LIN {X 0,Y 573.232,Z 251.703,A -85,B 0,C 180,E1 -2309.118,E2 -2309.118} C_VEL
LIN {X 0,Y 573.231,Z 251.702,A -85,B 0,C 180,E1 -2311.435,E2 -2311.435} C_VEL
LIN {X 0,Y 573.254,Z 251.705,A -85,B 0,C 180,E1 -2314.59,E2 -2314.59} C_VEL
LIN {X 0,Y 573.236,Z 251.705,A -85,B 0,C 180,E1 -2317.662,E2 -2317.662} C_VEL
LIN {X 0,Y 573.276,Z 251.851,A -85,B 0,C 180,E1 -2318.673,E2 -2318.673} C_VEL
LIN {X 0,Y 573.837,Z 256.408,A -85,B 0,C 180,E1 -2319.383,E2 -2319.383} C_VEL
LIN {X 0,Y 573.742,Z 263.76,A -85,B 0,C 180,E1 -2320.45,E2 -2320.45} C_VEL
LIN {X 0,Y 575.209,Z 270.767,A -85,B 0,C 180,E1 -2320.593,E2 -2320.593} C_VEL
LIN {X 0,Y 574.754,Z 427.05,A -85,B 0,C 180,E1 -2322.612,E2 -2322.612} C_VEL
LIN {X 0,Y 574.651,Z 442.817,A -85,B 0,C 180,E1 -2322.954,E2 -2322.954} C_VEL
LIN {X 0,Y 574.452,Z 456.451,A -85,B 0,C 180,E1 -2323.382,E2 -2323.382} C_VEL
LIN {X 0,Y 574.308,Z 469.862,A -85,B 0,C 180,E1 -2323.926,E2 -2323.926} C_VEL
LIN {X 0,Y 574.101,Z 483.847,A -85,B 0,C 180,E1 -2324.649,E2 -2324.649} C_VEL
LIN {X 0,Y 573.911,Z 496.092,A -85,B 0,C 180,E1 -2325.413,E2 -2325.413} C_VEL
LIN {X 0,Y 573.693,Z 508.609,A -85,B 0,C 180,E1 -2326.36,E2 -2326.36} C_VEL
LIN {X 0,Y 573.571,Z 518.669,A -85,B 0,C 180,E1 -2327.258,E2 -2327.258} C_VEL
LIN {X 0,Y 573.399,Z 528.984,A -85,B 0,C 180,E1 -2328.332,E2 -2328.332} C_VEL
LIN {X 0,Y 573.267,Z 538.996,A -85,B 0,C 180,E1 -2329.582,E2 -2329.582} C_VEL
LIN {X 0,Y 573.137,Z 547.362,A -85,B 0,C 180,E1 -2330.827,E2 -2330.827} C_VEL
LIN {X 0,Y 573.081,Z 555.183,A -85,B 0,C 180,E1 -2332.247,E2 -2332.247} C_VEL
LIN {X 0,Y 573.03,Z 561.427,A -85,B 0,C 180,E1 -2333.662,E2 -2333.662} C_VEL
LIN {X 0,Y 572.95,Z 566.262,A -85,B 0,C 180,E1 -2335.074,E2 -2335.074} C_VEL
LIN {X 0,Y 573.006,Z 569.794,A -85,B 0,C 180,E1 -2336.484,E2 -2336.484} C_VEL
LIN {X 0,Y 572.933,Z 572.153,A -85,B 0,C 180,E1 -2337.891,E2 -2337.891} C_VEL
LIN {X 0,Y 572.937,Z 573.314,A -85,B 0,C 180,E1 -2339.297,E2 -2339.297} C_VEL
LIN {X 0,Y 572.939,Z 573.342,A -85,B 0,C 180,E1 -2340.702,E2 -2340.702} C_VEL
LIN {X 0,Y 572.937,Z 572.256,A -85,B 0,C 180,E1 -2342.108,E2 -2342.108} C_VEL
LIN {X 0,Y 573.007,Z 569.983,A -85,B 0,C 180,E1 -2343.515,E2 -2343.515} C_VEL
LIN {X 0,Y 572.952,Z 566.528,A -85,B 0,C 180,E1 -2344.925,E2 -2344.925} C_VEL
LIN {X 0,Y 573.017,Z 561.792,A -85,B 0,C 180,E1 -2346.337,E2 -2346.337} C_VEL
LIN {X 0,Y 573.072,Z 555.625,A -85,B 0,C 180,E1 -2347.752,E2 -2347.752} C_VEL
LIN {X 0,Y 573.135,Z 547.941,A -85,B 0,C 180,E1 -2349.172,E2 -2349.172} C_VEL
LIN {X 0,Y 573.265,Z 539.657,A -85,B 0,C 180,E1 -2350.417,E2 -2350.417} C_VEL
LIN {X 0,Y 573.354,Z 529.786,A -85,B 0,C 180,E1 -2351.668,E2 -2351.668} C_VEL
LIN {X 0,Y 573.533,Z 519.618,A -85,B 0,C 180,E1 -2352.742,E2 -2352.742} C_VEL
LIN {X 0,Y 573.694,Z 508.608,A -85,B 0,C 180,E1 -2353.73,E2 -2353.73} C_VEL
LIN {X 0,Y 573.916,Z 496.248,A -85,B 0,C 180,E1 -2354.667,E2 -2354.667} C_VEL
LIN {X 0,Y 574.088,Z 483.851,A -85,B 0,C 180,E1 -2355.441,E2 -2355.441} C_VEL
LIN {X 0,Y 574.302,Z 469.864,A -85,B 0,C 180,E1 -2356.164,E2 -2356.164} C_VEL
LIN {X 0,Y 574.468,Z 456.434,A -85,B 0,C 180,E1 -2356.707,E2 -2356.707} C_VEL
LIN {X 0,Y 574.632,Z 441.329,A -85,B 0,C 180,E1 -2357.178,E2 -2357.178} C_VEL
LIN {X 0,Y 574.721,Z 432.945,A -85,B 0,C 180,E1 -2357.369,E2 -2357.369} C_VEL
LIN {X 0,Y 574.195,Z 427.214,A -85,B 0,C 180,E1 -2357.501,E2 -2357.501} C_VEL
LIN {X 0,Y 568.693,Z 408.639,A -85,B 0,C 180,E1 -2357.931,E2 -2357.931} C_VEL
LIN {X 0,Y 568.057,Z 402.835,A -85,B 0,C 180,E1 -2358.024,E2 -2358.024} C_VEL
LIN {X 0,Y 568.401,Z 270.982,A -85,B 0,C 180,E1 -2359.737,E2 -2359.737} C_VEL
LIN {X 0,Y 566.817,Z 263.453,A -85,B 0,C 180,E1 -2359.902,E2 -2359.902} C_VEL
LIN {X 0,Y 566.779,Z 255.764,A -85,B 0,C 180,E1 -2361.075,E2 -2361.075} C_VEL
LIN {X 0,Y 566.19,Z 252.586,A -85,B 0,C 180,E1 -2361.605,E2 -2361.605} C_VEL
LIN {X 0,Y 566.175,Z 252.587,A -85,B 0,C 180,E1 -2364.181,E2 -2364.181} C_VEL
LIN {X 0,Y 566.185,Z 252.579,A -85,B 0,C 180,E1 -2366.653,E2 -2366.653} C_VEL
LIN {X 0,Y 566.177,Z 252.579,A -85,B 0,C 180,E1 -2368.953,E2 -2368.953} C_VEL
LIN {X 0,Y 566.189,Z 252.58,A -85,B 0,C 180,E1 -2371.421,E2 -2371.421} C_VEL
LIN {X 0,Y 566.208,Z 252.584,A -85,B 0,C 180,E1 -2373.955,E2 -2373.955} C_VEL
LIN {X 0,Y 566.181,Z 252.579,A -85,B 0,C 180,E1 -2376.57,E2 -2376.57} C_VEL
LIN {X 0,Y 566.213,Z 252.581,A -85,B 0,C 180,E1 -2379.685,E2 -2379.685} C_VEL
LIN {X 0,Y 566.198,Z 252.576,A -85,B 0,C 180,E1 -2382.916,E2 -2382.916} C_VEL
LIN {X 0,Y 566.191,Z 252.583,A -85,B 0,C 180,E1 -2386.048,E2 -2386.048} C_VEL
LIN {X 0,Y 566.201,Z 252.577,A -85,B 0,C 180,E1 -2389.213,E2 -2389.213} C_VEL
LIN {X 0,Y 566.182,Z 252.586,A -85,B 0,C 180,E1 -2391.636,E2 -2391.636} C_VEL
LIN {X 0,Y 566.16,Z 252.583,A -85,B 0,C 180,E1 -2394.307,E2 -2394.307} C_VEL
LIN {X 0,Y 566.2,Z 252.576,A -85,B 0,C 180,E1 -2396.896,E2 -2396.896} C_VEL
LIN {X 0,Y 566.175,Z 252.584,A -85,B 0,C 180,E1 -2399.406,E2 -2399.406} C_VEL
LIN {X 0,Y 566.181,Z 252.586,A -85,B 0,C 180,E1 -2401.855,E2 -2401.855} C_VEL
LIN {X 0,Y 566.2,Z 252.578,A -85,B 0,C 180,E1 -2404.25,E2 -2404.25} C_VEL
LIN {X 0,Y 566.163,Z 252.58,A -85,B 0,C 180,E1 -2406.718,E2 -2406.718} C_VEL
LIN {X 0,Y 566.202,Z 252.586,A -85,B 0,C 180,E1 -2409.662,E2 -2409.662} C_VEL
LIN {X 0,Y 566.192,Z 252.577,A -85,B 0,C 180,E1 -2412.667,E2 -2412.667} C_VEL
LIN {X 0,Y 566.221,Z 252.583,A -85,B 0,C 180,E1 -2415.626,E2 -2415.626} C_VEL
LIN {X 0,Y 566.228,Z 252.572,A -85,B 0,C 180,E1 -2418.674,E2 -2418.674} C_VEL
LIN {X 0,Y 566.223,Z 252.58,A -85,B 0,C 180,E1 -2421.433,E2 -2421.433} C_VEL
LIN {X 0,Y 566.244,Z 252.571,A -85,B 0,C 180,E1 -2424.301,E2 -2424.301} C_VEL
LIN {X 0,Y 566.268,Z 252.571,A -85,B 0,C 180,E1 -2427.153,E2 -2427.153} C_VEL
LIN {X 0,Y 566.273,Z 252.57,A -85,B 0,C 180,E1 -2429.999,E2 -2429.999} C_VEL
LIN {X 0,Y 566.262,Z 252.569,A -85,B 0,C 180,E1 -2432.845,E2 -2432.845} C_VEL
LIN {X 0,Y 566.249,Z 252.577,A -85,B 0,C 180,E1 -2435.697,E2 -2435.697} C_VEL
LIN {X 0,Y 566.195,Z 252.576,A -85,B 0,C 180,E1 -2438.565,E2 -2438.565} C_VEL
LIN {X 0,Y 566.231,Z 252.582,A -85,B 0,C 180,E1 -2441.453,E2 -2441.453} C_VEL
LIN {X 0,Y 566.218,Z 252.573,A -85,B 0,C 180,E1 -2444.504,E2 -2444.504} C_VEL
LIN {X 0,Y 566.187,Z 252.585,A -85,B 0,C 180,E1 -2447.331,E2 -2447.331} C_VEL
LIN {X 0,Y 566.2,Z 252.576,A -85,B 0,C 180,E1 -2450.336,E2 -2450.336} C_VEL
LIN {X 0,Y 566.159,Z 252.589,A -85,B 0,C 180,E1 -2453.281,E2 -2453.281} C_VEL
LIN {X 0,Y 566.2,Z 252.58,A -85,B 0,C 180,E1 -2455.748,E2 -2455.748} C_VEL
LIN {X 0,Y 566.189,Z 252.577,A -85,B 0,C 180,E1 -2458.201,E2 -2458.201} C_VEL
LIN {X 0,Y 566.186,Z 252.583,A -85,B 0,C 180,E1 -2461.077,E2 -2461.077} C_VEL
LIN {X 0,Y 566.198,Z 252.58,A -85,B 0,C 180,E1 -2463.734,E2 -2463.734} C_VEL
LIN {X 0,Y 566.194,Z 252.577,A -85,B 0,C 180,E1 -2466.569,E2 -2466.569} C_VEL
LIN {X 0,Y 566.198,Z 252.58,A -85,B 0,C 180,E1 -2469.685,E2 -2469.685} C_VEL
LIN {X 0,Y 566.175,Z 252.579,A -85,B 0,C 180,E1 -2472.089,E2 -2472.089} C_VEL
LIN {X 0,Y 566.159,Z 252.587,A -85,B 0,C 180,E1 -2475.035,E2 -2475.035} C_VEL
LIN {X 0,Y 566.175,Z 252.58,A -85,B 0,C 180,E1 -2477.91,E2 -2477.91} C_VEL
LIN {X 0,Y 566.206,Z 252.577,A -85,B 0,C 180,E1 -2480.727,E2 -2480.727} C_VEL
LIN {X 0,Y 566.188,Z 252.579,A -85,B 0,C 180,E1 -2483.785,E2 -2483.785} C_VEL
LIN {X 0,Y 566.197,Z 252.576,A -85,B 0,C 180,E1 -2486.266,E2 -2486.266} C_VEL
LIN {X 0,Y 566.184,Z 252.583,A -85,B 0,C 180,E1 -2488.922,E2 -2488.922} C_VEL
LIN {X 0,Y 566.196,Z 252.577,A -85,B 0,C 180,E1 -2491.857,E2 -2491.857} C_VEL
LIN {X 0,Y 566.199,Z 252.576,A -85,B 0,C 180,E1 -2494.251,E2 -2494.251} C_VEL
LIN {X 0,Y 566.158,Z 252.584,A -85,B 0,C 180,E1 -2496.718,E2 -2496.718} C_VEL
LIN {X 0,Y 566.203,Z 252.578,A -85,B 0,C 180,E1 -2499.663,E2 -2499.663} C_VEL
LIN {X 0,Y 566.184,Z 252.581,A -85,B 0,C 180,E1 -2502.669,E2 -2502.669} C_VEL
LIN {X 0,Y 566.214,Z 252.576,A -85,B 0,C 180,E1 -2505.627,E2 -2505.627} C_VEL
LIN {X 0,Y 566.22,Z 252.577,A -85,B 0,C 180,E1 -2508.676,E2 -2508.676} C_VEL
LIN {X 0,Y 566.193,Z 252.581,A -85,B 0,C 180,E1 -2511.434,E2 -2511.434} C_VEL
LIN {X 0,Y 566.246,Z 252.571,A -85,B 0,C 180,E1 -2514.302,E2 -2514.302} C_VEL
LIN {X 0,Y 566.258,Z 252.569,A -85,B 0,C 180,E1 -2517.867,E2 -2517.867} C_VEL
LIN {X 0,Y 566.298,Z 252.569,A -85,B 0,C 180,E1 -2520.712,E2 -2520.712} C_VEL
LIN {X 0,Y 566.267,Z 252.575,A -85,B 0,C 180,E1 -2522.846,E2 -2522.846} C_VEL
LIN {X 0,Y 566.239,Z 252.572,A -85,B 0,C 180,E1 -2525.699,E2 -2525.699} C_VEL
LIN {X 0,Y 566.22,Z 252.577,A -85,B 0,C 180,E1 -2528.566,E2 -2528.566} C_VEL
LIN {X 0,Y 566.232,Z 252.574,A -85,B 0,C 180,E1 -2531.455,E2 -2531.455} C_VEL
LIN {X 0,Y 566.221,Z 252.577,A -85,B 0,C 180,E1 -2534.507,E2 -2534.507} C_VEL
LIN {X 0,Y 566.188,Z 252.581,A -85,B 0,C 180,E1 -2537.332,E2 -2537.332} C_VEL
LIN {X 0,Y 566.202,Z 252.577,A -85,B 0,C 180,E1 -2540.338,E2 -2540.338} C_VEL
LIN {X 0,Y 566.163,Z 252.584,A -85,B 0,C 180,E1 -2543.283,E2 -2543.283} C_VEL
LIN {X 0,Y 566.196,Z 252.576,A -85,B 0,C 180,E1 -2545.75,E2 -2545.75} C_VEL
LIN {X 0,Y 566.192,Z 252.578,A -85,B 0,C 180,E1 -2548.203,E2 -2548.203} C_VEL
LIN {X 0,Y 566.181,Z 252.584,A -85,B 0,C 180,E1 -2551.078,E2 -2551.078} C_VEL
LIN {X 0,Y 566.202,Z 252.576,A -85,B 0,C 180,E1 -2553.735,E2 -2553.735} C_VEL
LIN {X 0,Y 566.19,Z 252.583,A -85,B 0,C 180,E1 -2556.571,E2 -2556.571} C_VEL
LIN {X 0,Y 566.205,Z 252.575,A -85,B 0,C 180,E1 -2559.687,E2 -2559.687} C_VEL
LIN {X 0,Y 566.201,Z 252.577,A -85,B 0,C 180,E1 -2562.089,E2 -2562.089} C_VEL
LIN {X 0,Y 566.16,Z 252.586,A -85,B 0,C 180,E1 -2565.037,E2 -2565.037} C_VEL
LIN {X 0,Y 566.18,Z 252.579,A -85,B 0,C 180,E1 -2567.911,E2 -2567.911} C_VEL
LIN {X 0,Y 566.212,Z 252.585,A -85,B 0,C 180,E1 -2570.728,E2 -2570.728} C_VEL
LIN {X 0,Y 566.16,Z 252.581,A -85,B 0,C 180,E1 -2573.792,E2 -2573.792} C_VEL
LIN {X 0,Y 566.206,Z 252.579,A -85,B 0,C 180,E1 -2576.267,E2 -2576.267} C_VEL
LIN {X 0,Y 566.186,Z 252.585,A -85,B 0,C 180,E1 -2578.925,E2 -2578.925} C_VEL
LIN {X 0,Y 566.186,Z 252.583,A -85,B 0,C 180,E1 -2581.857,E2 -2581.857} C_VEL
LIN {X 0,Y 566.238,Z 252.628,A -85,B 0,C 180,E1 -2582.162,E2 -2582.162} C_VEL
LIN {X 0,Y 568.1,Z 261.431,A -85,B 0,C 180,E1 -2583.285,E2 -2583.285} C_VEL
LIN {X 0,Y 567.73,Z 286.752,A -85,B 0,C 180,E1 -2586.194,E2 -2586.194} C_VEL
LIN {X 0,Y 567.32,Z 312.6,A -85,B 0,C 180,E1 -2589.137,E2 -2589.137} C_VEL
LIN {X 0,Y 567.151,Z 321.407,A -85,B 0,C 180,E1 -2590.131,E2 -2590.131} C_VEL
LIN {X 0,Y 568.518,Z 329.423,A -85,B 0,C 180,E1 -2590.292,E2 -2590.292} C_VEL
LIN {X 0,Y 567.995,Z 488.204,A -85,B 0,C 180,E1 -2592.369,E2 -2592.369} C_VEL
LIN {X 0,Y 567.831,Z 503.746,A -85,B 0,C 180,E1 -2592.721,E2 -2592.721} C_VEL
LIN {X 0,Y 567.597,Z 519.068,A -85,B 0,C 180,E1 -2593.224,E2 -2593.224} C_VEL
LIN {X 0,Y 567.444,Z 532.799,A -85,B 0,C 180,E1 -2593.82,E2 -2593.82} C_VEL
LIN {X 0,Y 567.15,Z 546.267,A -85,B 0,C 180,E1 -2594.55,E2 -2594.55} C_VEL
LIN {X 0,Y 566.933,Z 558.519,A -85,B 0,C 180,E1 -2595.359,E2 -2595.359} C_VEL
LIN {X 0,Y 566.671,Z 571.305,A -85,B 0,C 180,E1 -2596.372,E2 -2596.372} C_VEL
LIN {X 0,Y 566.49,Z 582.76,A -85,B 0,C 180,E1 -2597.462,E2 -2597.462} C_VEL
LIN {X 0,Y 566.267,Z 593.32,A -85,B 0,C 180,E1 -2598.66,E2 -2598.66} C_VEL
LIN {X 0,Y 566.208,Z 601.864,A -85,B 0,C 180,E1 -2599.813,E2 -2599.813} C_VEL
LIN {X 0,Y 566.057,Z 609.74,A -85,B 0,C 180,E1 -2601.073,E2 -2601.073} C_VEL
LIN {X 0,Y 565.997,Z 617.094,A -85,B 0,C 180,E1 -2602.51,E2 -2602.51} C_VEL
LIN {X 0,Y 565.956,Z 622.926,A -85,B 0,C 180,E1 -2603.942,E2 -2603.942} C_VEL
LIN {X 0,Y 565.866,Z 626.389,A -85,B 0,C 180,E1 -2605.013,E2 -2605.013} C_VEL
LIN {X 0,Y 565.909,Z 629.892,A -85,B 0,C 180,E1 -2606.441,E2 -2606.441} C_VEL
LIN {X 0,Y 565.838,Z 632.193,A -85,B 0,C 180,E1 -2607.866,E2 -2607.866} C_VEL
LIN {X 0,Y 565.839,Z 633.349,A -85,B 0,C 180,E1 -2609.289,E2 -2609.289} C_VEL
LIN {X 0,Y 565.839,Z 633.348,A -85,B 0,C 180,E1 -2610.713,E2 -2610.713} C_VEL
LIN {X 0,Y 565.838,Z 632.189,A -85,B 0,C 180,E1 -2612.136,E2 -2612.136} C_VEL
LIN {X 0,Y 565.909,Z 629.885,A -85,B 0,C 180,E1 -2613.561,E2 -2613.561} C_VEL
LIN {X 0,Y 565.867,Z 626.383,A -85,B 0,C 180,E1 -2614.988,E2 -2614.988} C_VEL
LIN {X 0,Y 565.956,Z 622.922,A -85,B 0,C 180,E1 -2616.06,E2 -2616.06} C_VEL
LIN {X 0,Y 565.999,Z 617.084,A -85,B 0,C 180,E1 -2617.492,E2 -2617.492} C_VEL
LIN {X 0,Y 566.058,Z 609.726,A -85,B 0,C 180,E1 -2618.929,E2 -2618.929} C_VEL
LIN {X 0,Y 566.209,Z 601.85,A -85,B 0,C 180,E1 -2620.189,E2 -2620.189} C_VEL
LIN {X 0,Y 566.311,Z 592.383,A -85,B 0,C 180,E1 -2621.454,E2 -2621.454} C_VEL
LIN {X 0,Y 566.492,Z 582.74,A -85,B 0,C 180,E1 -2622.54,E2 -2622.54} C_VEL
LIN {X 0,Y 566.671,Z 571.285,A -85,B 0,C 180,E1 -2623.63,E2 -2623.63} C_VEL
LIN {X 0,Y 566.93,Z 558.666,A -85,B 0,C 180,E1 -2624.631,E2 -2624.631} C_VEL
LIN {X 0,Y 567.149,Z 546.231,A -85,B 0,C 180,E1 -2625.452,E2 -2625.452} C_VEL
LIN {X 0,Y 567.46,Z 532.75,A -85,B 0,C 180,E1 -2626.181,E2 -2626.181} C_VEL
LIN {X 0,Y 567.617,Z 519.025,A -85,B 0,C 180,E1 -2626.778,E2 -2626.778} C_VEL
LIN {X 0,Y 567.85,Z 503.688,A -85,B 0,C 180,E1 -2627.28,E2 -2627.28} C_VEL
LIN {X 0,Y 567.984,Z 488.256,A -85,B 0,C 180,E1 -2627.63,E2 -2627.63} C_VEL
LIN {X 0,Y 568.475,Z 328.292,A -85,B 0,C 180,E1 -2629.725,E2 -2629.725} C_VEL
LIN {X 0,Y 567.151,Z 321.264,A -85,B 0,C 180,E1 -2629.885,E2 -2629.885} C_VEL
LIN {X 0,Y 567.556,Z 297.587,A -85,B 0,C 180,E1 -2632.574,E2 -2632.574} C_VEL
LIN {X 0,Y 567.871,Z 272.563,A -85,B 0,C 180,E1 -2635.384,E2 -2635.384} C_VEL
LIN {X 0,Y 567.957,Z 260.783,A -85,B 0,C 180,E1 -2636.721,E2 -2636.721} C_VEL
LIN {X 0,Y 566.229,Z 252.58,A -85,B 0,C 180,E1 -2637.74,E2 -2637.74} C_VEL
LIN {X 0,Y 566.177,Z 252.583,A -85,B 0,C 180,E1 -2640.594,E2 -2640.594} C_VEL
LIN {X 0,Y 566.215,Z 252.585,A -85,B 0,C 180,E1 -2643.103,E2 -2643.103} C_VEL
LIN {X 0,Y 566.166,Z 252.584,A -85,B 0,C 180,E1 -2645.693,E2 -2645.693} C_VEL
LIN {X 0,Y 566.217,Z 252.579,A -85,B 0,C 180,E1 -2648.559,E2 -2648.559} C_VEL
LIN {X 0,Y 566.177,Z 252.587,A -85,B 0,C 180,E1 -2651.14,E2 -2651.14} C_VEL
LIN {X 0,Y 566.197,Z 252.578,A -85,B 0,C 180,E1 -2654.037,E2 -2654.037} C_VEL
LIN {X 0,Y 566.208,Z 252.581,A -85,B 0,C 180,E1 -2657.083,E2 -2657.083} C_VEL
LIN {X 0,Y 566.218,Z 252.579,A -85,B 0,C 180,E1 -2660.315,E2 -2660.315} C_VEL
LIN {X 0,Y 566.187,Z 252.579,A -85,B 0,C 180,E1 -2663.429,E2 -2663.429} C_VEL
LIN {X 0,Y 566.217,Z 252.581,A -85,B 0,C 180,E1 -2666.266,E2 -2666.266} C_VEL
LIN {X 0,Y 566.195,Z 252.581,A -85,B 0,C 180,E1 -2668.924,E2 -2668.924} C_VEL
LIN {X 0,Y 566.192,Z 252.582,A -85,B 0,C 180,E1 -2671.856,E2 -2671.856} C_VEL
LIN {X 0,Y 566.215,Z 252.584,A -85,B 0,C 180,E1 -2674.251,E2 -2674.251} C_VEL
LIN {X 0,Y 566.173,Z 252.586,A -85,B 0,C 180,E1 -2676.719,E2 -2676.719} C_VEL
LIN {X 0,Y 566.239,Z 252.773,A -85,B 0,C 180,E1 -2678.515,E2 -2678.515} C_VEL
LIN {X 0,Y 566.905,Z 257.656,A -85,B 0,C 180,E1 -2679.309,E2 -2679.309} C_VEL
LIN {X 0,Y 566.766,Z 263.49,A -85,B 0,C 180,E1 -2680.192,E2 -2680.192} C_VEL
LIN {X 0,Y 568.445,Z 271.097,A -85,B 0,C 180,E1 -2680.356,E2 -2680.356} C_VEL
LIN {X 0,Y 567.99,Z 427.142,A -85,B 0,C 180,E1 -2682.4,E2 -2682.4} C_VEL
LIN {X 0,Y 567.873,Z 442.816,A -85,B 0,C 180,E1 -2682.744,E2 -2682.744} C_VEL
LIN {X 0,Y 567.638,Z 456.453,A -85,B 0,C 180,E1 -2683.177,E2 -2683.177} C_VEL
LIN {X 0,Y 567.451,Z 469.884,A -85,B 0,C 180,E1 -2683.727,E2 -2683.727} C_VEL
LIN {X 0,Y 567.222,Z 483.85,A -85,B 0,C 180,E1 -2684.458,E2 -2684.458} C_VEL
LIN {X 0,Y 566.969,Z 496.677,A -85,B 0,C 180,E1 -2685.27,E2 -2685.27} C_VEL
LIN {X 0,Y 566.728,Z 509.669,A -85,B 0,C 180,E1 -2686.28,E2 -2686.28} C_VEL
LIN {X 0,Y 566.552,Z 520.536,A -85,B 0,C 180,E1 -2687.28,E2 -2687.28} C_VEL
LIN {X 0,Y 566.314,Z 532.007,A -85,B 0,C 180,E1 -2688.547,E2 -2688.547} C_VEL
LIN {X 0,Y 566.214,Z 541.564,A -85,B 0,C 180,E1 -2689.812,E2 -2689.812} C_VEL
LIN {X 0,Y 566.059,Z 549.473,A -85,B 0,C 180,E1 -2691.071,E2 -2691.071} C_VEL
LIN {X 0,Y 565.995,Z 556.893,A -85,B 0,C 180,E1 -2692.508,E2 -2692.508} C_VEL
LIN {X 0,Y 565.96,Z 562.764,A -85,B 0,C 180,E1 -2693.941,E2 -2693.941} C_VEL
LIN {X 0,Y 565.866,Z 566.267,A -85,B 0,C 180,E1 -2695.012,E2 -2695.012} C_VEL
LIN {X 0,Y 565.911,Z 569.789,A -85,B 0,C 180,E1 -2696.439,E2 -2696.439} C_VEL
LIN {X 0,Y 565.835,Z 572.156,A -85,B 0,C 180,E1 -2697.864,E2 -2697.864} C_VEL
LIN {X 0,Y 565.837,Z 573.309,A -85,B 0,C 180,E1 -2699.288,E2 -2699.288} C_VEL
LIN {X 0,Y 565.839,Z 573.337,A -85,B 0,C 180,E1 -2700.711,E2 -2700.711} C_VEL
LIN {X 0,Y 565.838,Z 572.258,A -85,B 0,C 180,E1 -2702.135,E2 -2702.135} C_VEL
LIN {X 0,Y 565.912,Z 569.983,A -85,B 0,C 180,E1 -2703.559,E2 -2703.559} C_VEL
LIN {X 0,Y 565.867,Z 566.52,A -85,B 0,C 180,E1 -2704.987,E2 -2704.987} C_VEL
LIN {X 0,Y 565.946,Z 561.79,A -85,B 0,C 180,E1 -2706.416,E2 -2706.416} C_VEL
LIN {X 0,Y 565.997,Z 555.615,A -85,B 0,C 180,E1 -2707.85,E2 -2707.85} C_VEL
LIN {X 0,Y 566.07,Z 547.937,A -85,B 0,C 180,E1 -2709.288,E2 -2709.288} C_VEL
LIN {X 0,Y 566.239,Z 539.645,A -85,B 0,C 180,E1 -2710.548,E2 -2710.548} C_VEL
LIN {X 0,Y 566.33,Z 529.781,A -85,B 0,C 180,E1 -2711.815,E2 -2711.815} C_VEL
LIN {X 0,Y 566.532,Z 519.602,A -85,B 0,C 180,E1 -2712.902,E2 -2712.902} C_VEL
LIN {X 0,Y 566.74,Z 508.596,A -85,B 0,C 180,E1 -2713.901,E2 -2713.901} C_VEL
LIN {X 0,Y 567,Z 496.081,A -85,B 0,C 180,E1 -2714.86,E2 -2714.86} C_VEL
LIN {X 0,Y 567.19,Z 483.835,A -85,B 0,C 180,E1 -2715.634,E2 -2715.634} C_VEL
LIN {X 0,Y 567.474,Z 469.862,A -85,B 0,C 180,E1 -2716.364,E2 -2716.364} C_VEL
LIN {X 0,Y 567.662,Z 456.403,A -85,B 0,C 180,E1 -2716.914,E2 -2716.914} C_VEL
LIN {X 0,Y 567.838,Z 441.713,A -85,B 0,C 180,E1 -2717.379,E2 -2717.379} C_VEL
LIN {X 0,Y 567.987,Z 426.978,A -85,B 0,C 180,E1 -2717.693,E2 -2717.693} C_VEL
LIN {X 0,Y 568.057,Z 402.835,A -85,B 0,C 180,E1 -2718.024,E2 -2718.024} C_VEL
LIN {X 0,Y 567.439,Z 397.035,A -85,B 0,C 180,E1 -2718.12,E2 -2718.12} C_VEL
LIN {X 0,Y 562.026,Z 378.413,A -85,B 0,C 180,E1 -2718.546,E2 -2718.546} C_VEL
LIN {X 0,Y 561.442,Z 372.613,A -85,B 0,C 180,E1 -2718.642,E2 -2718.642} C_VEL
LIN {X 0,Y 561.683,Z 271.819,A -85,B 0,C 180,E1 -2719.971,E2 -2719.971} C_VEL
LIN {X 0,Y 559.9,Z 263.572,A -85,B 0,C 180,E1 -2720.154,E2 -2720.154} C_VEL
LIN {X 0,Y 559.881,Z 257.225,A -85,B 0,C 180,E1 -2721.154,E2 -2721.154} C_VEL
LIN {X 0,Y 559.158,Z 253.463,A -85,B 0,C 180,E1 -2721.814,E2 -2721.814} C_VEL
LIN {X 0,Y 559.125,Z 253.461,A -85,B 0,C 180,E1 -2724.506,E2 -2724.506} C_VEL
LIN {X 0,Y 559.158,Z 253.454,A -85,B 0,C 180,E1 -2726.902,E2 -2726.902} C_VEL
LIN {X 0,Y 559.138,Z 253.465,A -85,B 0,C 180,E1 -2729.855,E2 -2729.855} C_VEL
LIN {X 0,Y 559.155,Z 253.454,A -85,B 0,C 180,E1 -2732.714,E2 -2732.714} C_VEL
LIN {X 0,Y 559.122,Z 253.46,A -85,B 0,C 180,E1 -2735.323,E2 -2735.323} C_VEL
LIN {X 0,Y 559.128,Z 253.464,A -85,B 0,C 180,E1 -2738.017,E2 -2738.017} C_VEL
LIN {X 0,Y 559.153,Z 253.454,A -85,B 0,C 180,E1 -2740.812,E2 -2740.812} C_VEL
LIN {X 0,Y 559.138,Z 253.464,A -85,B 0,C 180,E1 -2743.733,E2 -2743.733} C_VEL
LIN {X 0,Y 559.14,Z 253.455,A -85,B 0,C 180,E1 -2746.803,E2 -2746.803} C_VEL
LIN {X 0,Y 559.153,Z 253.455,A -85,B 0,C 180,E1 -2749.187,E2 -2749.187} C_VEL
LIN {X 0,Y 559.129,Z 253.463,A -85,B 0,C 180,E1 -2751.981,E2 -2751.981} C_VEL
LIN {X 0,Y 559.13,Z 253.456,A -85,B 0,C 180,E1 -2754.786,E2 -2754.786} C_VEL
LIN {X 0,Y 559.15,Z 253.458,A -85,B 0,C 180,E1 -2757.364,E2 -2757.364} C_VEL
LIN {X 0,Y 559.143,Z 253.458,A -85,B 0,C 180,E1 -2760.142,E2 -2760.142} C_VEL
LIN {X 0,Y 559.125,Z 253.459,A -85,B 0,C 180,E1 -2762.284,E2 -2762.284} C_VEL
LIN {X 0,Y 559.174,Z 253.451,A -85,B 0,C 180,E1 -2764.812,E2 -2764.812} C_VEL
LIN {X 0,Y 559.134,Z 253.463,A -85,B 0,C 180,E1 -2767.846,E2 -2767.846} C_VEL
LIN {X 0,Y 559.186,Z 253.45,A -85,B 0,C 180,E1 -2770.493,E2 -2770.493} C_VEL
LIN {X 0,Y 559.177,Z 253.454,A -85,B 0,C 180,E1 -2773.197,E2 -2773.197} C_VEL
LIN {X 0,Y 559.159,Z 253.455,A -85,B 0,C 180,E1 -2776.183,E2 -2776.183} C_VEL
LIN {X 0,Y 559.188,Z 253.452,A -85,B 0,C 180,E1 -2779.132,E2 -2779.132} C_VEL
LIN {X 0,Y 559.196,Z 253.451,A -85,B 0,C 180,E1 -2782.053,E2 -2782.053} C_VEL
LIN {X 0,Y 559.246,Z 253.443,A -85,B 0,C 180,E1 -2784.952,E2 -2784.952} C_VEL
LIN {X 0,Y 559.237,Z 253.449,A -85,B 0,C 180,E1 -2787.838,E2 -2787.838} C_VEL
LIN {X 0,Y 559.262,Z 253.44,A -85,B 0,C 180,E1 -2790.719,E2 -2790.719} C_VEL
LIN {X 0,Y 559.229,Z 253.445,A -85,B 0,C 180,E1 -2792.88,E2 -2792.88} C_VEL
LIN {X 0,Y 559.217,Z 253.452,A -85,B 0,C 180,E1 -2795.769,E2 -2795.769} C_VEL
LIN {X 0,Y 559.16,Z 253.453,A -85,B 0,C 180,E1 -2798.674,E2 -2798.674} C_VEL
LIN {X 0,Y 559.194,Z 253.457,A -85,B 0,C 180,E1 -2801.6,E2 -2801.6} C_VEL
LIN {X 0,Y 559.189,Z 253.449,A -85,B 0,C 180,E1 -2804.595,E2 -2804.595} C_VEL
LIN {X 0,Y 559.146,Z 253.463,A -85,B 0,C 180,E1 -2807.556,E2 -2807.556} C_VEL
LIN {X 0,Y 559.16,Z 253.457,A -85,B 0,C 180,E1 -2809.837,E2 -2809.837} C_VEL
LIN {X 0,Y 559.129,Z 253.457,A -85,B 0,C 180,E1 -2812.152,E2 -2812.152} C_VEL
LIN {X 0,Y 559.163,Z 253.461,A -85,B 0,C 180,E1 -2815.297,E2 -2815.297} C_VEL
LIN {X 0,Y 559.168,Z 253.457,A -85,B 0,C 180,E1 -2817.711,E2 -2817.711} C_VEL
LIN {X 0,Y 559.143,Z 253.455,A -85,B 0,C 180,E1 -2820.182,E2 -2820.182} C_VEL
LIN {X 0,Y 559.161,Z 253.454,A -85,B 0,C 180,E1 -2822.713,E2 -2822.713} C_VEL
LIN {X 0,Y 559.137,Z 253.466,A -85,B 0,C 180,E1 -2825.322,E2 -2825.322} C_VEL
LIN {X 0,Y 559.12,Z 253.459,A -85,B 0,C 180,E1 -2828.017,E2 -2828.017} C_VEL
LIN {X 0,Y 559.159,Z 253.455,A -85,B 0,C 180,E1 -2830.81,E2 -2830.81} C_VEL
LIN {X 0,Y 559.148,Z 253.458,A -85,B 0,C 180,E1 -2833.731,E2 -2833.731} C_VEL
LIN {X 0,Y 559.153,Z 253.456,A -85,B 0,C 180,E1 -2836.801,E2 -2836.801} C_VEL
LIN {X 0,Y 559.158,Z 253.462,A -85,B 0,C 180,E1 -2839.189,E2 -2839.189} C_VEL
LIN {X 0,Y 559.119,Z 253.459,A -85,B 0,C 180,E1 -2841.982,E2 -2841.982} C_VEL
LIN {X 0,Y 559.139,Z 253.459,A -85,B 0,C 180,E1 -2844.784,E2 -2844.784} C_VEL
LIN {X 0,Y 559.159,Z 253.46,A -85,B 0,C 180,E1 -2847.361,E2 -2847.361} C_VEL
LIN {X 0,Y 559.134,Z 253.456,A -85,B 0,C 180,E1 -2850.142,E2 -2850.142} C_VEL
LIN {X 0,Y 559.154,Z 253.462,A -85,B 0,C 180,E1 -2853.098,E2 -2853.098} C_VEL
LIN {X 0,Y 559.141,Z 253.46,A -85,B 0,C 180,E1 -2855.495,E2 -2855.495} C_VEL
LIN {X 0,Y 559.163,Z 253.455,A -85,B 0,C 180,E1 -2858.624,E2 -2858.624} C_VEL
LIN {X 0,Y 559.154,Z 253.46,A -85,B 0,C 180,E1 -2860.926,E2 -2860.926} C_VEL
LIN {X 0,Y 559.151,Z 253.454,A -85,B 0,C 180,E1 -2863.948,E2 -2863.948} C_VEL
LIN {X 0,Y 559.154,Z 253.453,A -85,B 0,C 180,E1 -2866.184,E2 -2866.184} C_VEL
LIN {X 0,Y 559.191,Z 253.452,A -85,B 0,C 180,E1 -2868.605,E2 -2868.605} C_VEL
LIN {X 0,Y 559.157,Z 253.459,A -85,B 0,C 180,E1 -2871.326,E2 -2871.326} C_VEL
LIN {X 0,Y 559.214,Z 253.446,A -85,B 0,C 180,E1 -2874.23,E2 -2874.23} C_VEL
LIN {X 0,Y 559.231,Z 253.444,A -85,B 0,C 180,E1 -2877.84,E2 -2877.84} C_VEL
LIN {X 0,Y 559.267,Z 253.445,A -85,B 0,C 180,E1 -2880.721,E2 -2880.721} C_VEL
LIN {X 0,Y 559.232,Z 253.452,A -85,B 0,C 180,E1 -2882.882,E2 -2882.882} C_VEL
LIN {X 0,Y 559.209,Z 253.447,A -85,B 0,C 180,E1 -2885.771,E2 -2885.771} C_VEL
LIN {X 0,Y 559.179,Z 253.456,A -85,B 0,C 180,E1 -2888.675,E2 -2888.675} C_VEL
LIN {X 0,Y 559.194,Z 253.45,A -85,B 0,C 180,E1 -2891.601,E2 -2891.601} C_VEL
LIN {X 0,Y 559.188,Z 253.454,A -85,B 0,C 180,E1 -2894.596,E2 -2894.596} C_VEL
LIN {X 0,Y 559.147,Z 253.456,A -85,B 0,C 180,E1 -2897.558,E2 -2897.558} C_VEL
LIN {X 0,Y 559.157,Z 253.453,A -85,B 0,C 180,E1 -2899.838,E2 -2899.838} C_VEL
LIN {X 0,Y 559.135,Z 253.457,A -85,B 0,C 180,E1 -2902.153,E2 -2902.153} C_VEL
LIN {X 0,Y 559.163,Z 253.456,A -85,B 0,C 180,E1 -2905.299,E2 -2905.299} C_VEL
LIN {X 0,Y 559.144,Z 253.455,A -85,B 0,C 180,E1 -2907.714,E2 -2907.714} C_VEL
LIN {X 0,Y 559.143,Z 253.456,A -85,B 0,C 180,E1 -2910.184,E2 -2910.184} C_VEL
LIN {X 0,Y 559.144,Z 253.463,A -85,B 0,C 180,E1 -2912.716,E2 -2912.716} C_VEL
LIN {X 0,Y 559.119,Z 253.46,A -85,B 0,C 180,E1 -2915.325,E2 -2915.325} C_VEL
LIN {X 0,Y 559.123,Z 253.458,A -85,B 0,C 180,E1 -2918.019,E2 -2918.019} C_VEL
LIN {X 0,Y 559.149,Z 253.464,A -85,B 0,C 180,E1 -2920.813,E2 -2920.813} C_VEL
LIN {X 0,Y 559.134,Z 253.459,A -85,B 0,C 180,E1 -2923.197,E2 -2923.197} C_VEL
LIN {X 0,Y 559.132,Z 253.459,A -85,B 0,C 180,E1 -2926.267,E2 -2926.267} C_VEL
LIN {X 0,Y 559.148,Z 253.458,A -85,B 0,C 180,E1 -2929.189,E2 -2929.189} C_VEL
LIN {X 0,Y 559.124,Z 253.459,A -85,B 0,C 180,E1 -2931.983,E2 -2931.983} C_VEL
LIN {X 0,Y 559.123,Z 253.466,A -85,B 0,C 180,E1 -2934.789,E2 -2934.789} C_VEL
LIN {X 0,Y 559.15,Z 253.456,A -85,B 0,C 180,E1 -2937.366,E2 -2937.366} C_VEL
LIN {X 0,Y 559.139,Z 253.46,A -85,B 0,C 180,E1 -2940.145,E2 -2940.145} C_VEL
LIN {X 0,Y 559.163,Z 253.564,A -85,B 0,C 180,E1 -2941.925,E2 -2941.925} C_VEL
LIN {X 0,Y 561.149,Z 261.791,A -85,B 0,C 180,E1 -2943.005,E2 -2943.005} C_VEL
LIN {X 0,Y 561.111,Z 273.623,A -85,B 0,C 180,E1 -2944.397,E2 -2944.397} C_VEL
LIN {X 0,Y 560.712,Z 297.365,A -85,B 0,C 180,E1 -2947.137,E2 -2947.137} C_VEL
LIN {X 0,Y 560.342,Z 321.738,A -85,B 0,C 180,E1 -2949.889,E2 -2949.889} C_VEL
LIN {X 0,Y 561.827,Z 329.762,A -85,B 0,C 180,E1 -2950.052,E2 -2950.052} C_VEL
LIN {X 0,Y 561.24,Z 488.288,A -85,B 0,C 180,E1 -2952.151,E2 -2952.151} C_VEL
LIN {X 0,Y 561.057,Z 503.744,A -85,B 0,C 180,E1 -2952.506,E2 -2952.506} C_VEL
LIN {X 0,Y 560.809,Z 519.065,A -85,B 0,C 180,E1 -2953.015,E2 -2953.015} C_VEL
LIN {X 0,Y 560.605,Z 532.802,A -85,B 0,C 180,E1 -2953.617,E2 -2953.617} C_VEL
LIN {X 0,Y 560.285,Z 546.27,A -85,B 0,C 180,E1 -2954.356,E2 -2954.356} C_VEL
LIN {X 0,Y 559.999,Z 559.304,A -85,B 0,C 180,E1 -2955.23,E2 -2955.23} C_VEL
LIN {X 0,Y 559.722,Z 571.306,A -85,B 0,C 180,E1 -2956.199,E2 -2956.199} C_VEL
LIN {X 0,Y 559.515,Z 582.76,A -85,B 0,C 180,E1 -2957.303,E2 -2957.303} C_VEL
LIN {X 0,Y 559.303,Z 592.398,A -85,B 0,C 180,E1 -2958.403,E2 -2958.403} C_VEL
LIN {X 0,Y 559.168,Z 601.863,A -85,B 0,C 180,E1 -2959.684,E2 -2959.684} C_VEL
LIN {X 0,Y 559.003,Z 609.741,A -85,B 0,C 180,E1 -2960.959,E2 -2960.959} C_VEL
LIN {X 0,Y 558.92,Z 617.095,A -85,B 0,C 180,E1 -2962.414,E2 -2962.414} C_VEL
LIN {X 0,Y 558.858,Z 622.926,A -85,B 0,C 180,E1 -2963.865,E2 -2963.865} C_VEL
LIN {X 0,Y 558.787,Z 626.389,A -85,B 0,C 180,E1 -2964.95,E2 -2964.95} C_VEL
LIN {X 0,Y 558.818,Z 629.891,A -85,B 0,C 180,E1 -2966.396,E2 -2966.396} C_VEL
LIN {X 0,Y 558.744,Z 632.192,A -85,B 0,C 180,E1 -2967.838,E2 -2967.838} C_VEL
LIN {X 0,Y 558.739,Z 633.349,A -85,B 0,C 180,E1 -2969.28,E2 -2969.28} C_VEL
LIN {X 0,Y 558.739,Z 633.348,A -85,B 0,C 180,E1 -2970.722,E2 -2970.722} C_VEL
LIN {X 0,Y 558.744,Z 632.188,A -85,B 0,C 180,E1 -2972.164,E2 -2972.164} C_VEL
LIN {X 0,Y 558.818,Z 629.884,A -85,B 0,C 180,E1 -2973.606,E2 -2973.606} C_VEL
LIN {X 0,Y 558.787,Z 626.383,A -85,B 0,C 180,E1 -2975.052,E2 -2975.052} C_VEL
LIN {X 0,Y 558.844,Z 621.605,A -85,B 0,C 180,E1 -2976.5,E2 -2976.5} C_VEL
LIN {X 0,Y 558.951,Z 615.417,A -85,B 0,C 180,E1 -2977.951,E2 -2977.951} C_VEL
LIN {X 0,Y 559.006,Z 607.64,A -85,B 0,C 180,E1 -2979.408,E2 -2979.408} C_VEL
LIN {X 0,Y 559.218,Z 599.361,A -85,B 0,C 180,E1 -2980.684,E2 -2980.684} C_VEL
LIN {X 0,Y 559.364,Z 589.384,A -85,B 0,C 180,E1 -2981.966,E2 -2981.966} C_VEL
LIN {X 0,Y 559.598,Z 579.178,A -85,B 0,C 180,E1 -2983.066,E2 -2983.066} C_VEL
LIN {X 0,Y 559.864,Z 567.009,A -85,B 0,C 180,E1 -2984.17,E2 -2984.17} C_VEL
LIN {X 0,Y 560.125,Z 554.676,A -85,B 0,C 180,E1 -2985.101,E2 -2985.101} C_VEL
LIN {X 0,Y 560.362,Z 541.494,A -85,B 0,C 180,E1 -2985.924,E2 -2985.924} C_VEL
LIN {X 0,Y 560.685,Z 526.807,A -85,B 0,C 180,E1 -2986.663,E2 -2986.663} C_VEL
LIN {X 0,Y 560.927,Z 512.591,A -85,B 0,C 180,E1 -2987.219,E2 -2987.219} C_VEL
LIN {X 0,Y 561.146,Z 498.116,A -85,B 0,C 180,E1 -2987.638,E2 -2987.638} C_VEL
LIN {X 0,Y 561.237,Z 483.588,A -85,B 0,C 180,E1 -2987.924,E2 -2987.924} C_VEL
LIN {X 0,Y 561.808,Z 329.437,A -85,B 0,C 180,E1 -2989.953,E2 -2989.953} C_VEL
LIN {X 0,Y 560.317,Z 321.397,A -85,B 0,C 180,E1 -2990.123,E2 -2990.123} C_VEL
LIN {X 0,Y 560.635,Z 298.799,A -85,B 0,C 180,E1 -2992.674,E2 -2992.674} C_VEL
LIN {X 0,Y 560.976,Z 274.216,A -85,B 0,C 180,E1 -2995.459,E2 -2995.459} C_VEL
LIN {X 0,Y 561.124,Z 262.508,A -85,B 0,C 180,E1 -2996.802,E2 -2996.802} C_VEL
LIN {X 0,Y 559.178,Z 253.457,A -85,B 0,C 180,E1 -2997.964,E2 -2997.964} C_VEL
LIN {X 0,Y 559.156,Z 253.463,A -85,B 0,C 180,E1 -3001.02,E2 -3001.02} C_VEL
LIN {X 0,Y 559.17,Z 253.455,A -85,B 0,C 180,E1 -3003.949,E2 -3003.949} C_VEL
LIN {X 0,Y 559.146,Z 253.464,A -85,B 0,C 180,E1 -3007.109,E2 -3007.109} C_VEL
LIN {X 0,Y 559.17,Z 253.454,A -85,B 0,C 180,E1 -3009.943,E2 -3009.943} C_VEL
LIN {X 0,Y 559.162,Z 253.462,A -85,B 0,C 180,E1 -3012.744,E2 -3012.744} C_VEL
LIN {X 0,Y 559.157,Z 253.455,A -85,B 0,C 180,E1 -3015.761,E2 -3015.761} C_VEL
LIN {X 0,Y 559.168,Z 253.456,A -85,B 0,C 180,E1 -3018.23,E2 -3018.23} C_VEL
LIN {X 0,Y 559.178,Z 253.454,A -85,B 0,C 180,E1 -3021.192,E2 -3021.192} C_VEL
LIN {X 0,Y 559.127,Z 253.459,A -85,B 0,C 180,E1 -3023.788,E2 -3023.788} C_VEL
LIN {X 0,Y 559.169,Z 253.462,A -85,B 0,C 180,E1 -3026.425,E2 -3026.425} C_VEL
LIN {X 0,Y 559.159,Z 253.457,A -85,B 0,C 180,E1 -3028.981,E2 -3028.981} C_VEL
LIN {X 0,Y 559.139,Z 253.459,A -85,B 0,C 180,E1 -3031.625,E2 -3031.625} C_VEL
LIN {X 0,Y 559.18,Z 253.457,A -85,B 0,C 180,E1 -3033.903,E2 -3033.903} C_VEL
LIN {X 0,Y 559.143,Z 253.464,A -85,B 0,C 180,E1 -3036.572,E2 -3036.572} C_VEL
LIN {X 0,Y 559.192,Z 253.637,A -85,B 0,C 180,E1 -3038.279,E2 -3038.279} C_VEL
LIN {X 0,Y 560.018,Z 258.086,A -85,B 0,C 180,E1 -3039.043,E2 -3039.043} C_VEL
LIN {X 0,Y 559.853,Z 263.713,A -85,B 0,C 180,E1 -3039.937,E2 -3039.937} C_VEL
LIN {X 0,Y 561.804,Z 273.348,A -85,B 0,C 180,E1 -3040.144,E2 -3040.144} C_VEL
LIN {X 0,Y 561.212,Z 427.312,A -85,B 0,C 180,E1 -3042.183,E2 -3042.183} C_VEL
LIN {X 0,Y 561.059,Z 443.602,A -85,B 0,C 180,E1 -3042.551,E2 -3042.551} C_VEL
LIN {X 0,Y 560.847,Z 456.455,A -85,B 0,C 180,E1 -3042.967,E2 -3042.967} C_VEL
LIN {X 0,Y 560.628,Z 469.905,A -85,B 0,C 180,E1 -3043.523,E2 -3043.523} C_VEL
LIN {X 0,Y 560.349,Z 483.852,A -85,B 0,C 180,E1 -3044.262,E2 -3044.262} C_VEL
LIN {X 0,Y 560.052,Z 496.551,A -85,B 0,C 180,E1 -3045.076,E2 -3045.076} C_VEL
LIN {X 0,Y 559.796,Z 508.614,A -85,B 0,C 180,E1 -3046.014,E2 -3046.014} C_VEL
LIN {X 0,Y 559.594,Z 518.661,A -85,B 0,C 180,E1 -3046.934,E2 -3046.934} C_VEL
LIN {X 0,Y 559.384,Z 528.995,A -85,B 0,C 180,E1 -3048.035,E2 -3048.035} C_VEL
LIN {X 0,Y 559.212,Z 538.988,A -85,B 0,C 180,E1 -3049.317,E2 -3049.317} C_VEL
LIN {X 0,Y 559.007,Z 547.367,A -85,B 0,C 180,E1 -3050.593,E2 -3050.593} C_VEL
LIN {X 0,Y 558.945,Z 555.174,A -85,B 0,C 180,E1 -3052.049,E2 -3052.049} C_VEL
LIN {X 0,Y 558.856,Z 561.259,A -85,B 0,C 180,E1 -3053.457,E2 -3053.457} C_VEL
LIN {X 0,Y 558.787,Z 566.267,A -85,B 0,C 180,E1 -3054.949,E2 -3054.949} C_VEL
LIN {X 0,Y 558.82,Z 569.785,A -85,B 0,C 180,E1 -3056.394,E2 -3056.394} C_VEL
LIN {X 0,Y 558.741,Z 572.159,A -85,B 0,C 180,E1 -3057.837,E2 -3057.837} C_VEL
LIN {X 0,Y 558.738,Z 573.305,A -85,B 0,C 180,E1 -3059.279,E2 -3059.279} C_VEL
LIN {X 0,Y 558.74,Z 573.332,A -85,B 0,C 180,E1 -3060.72,E2 -3060.72} C_VEL
LIN {X 0,Y 558.744,Z 572.26,A -85,B 0,C 180,E1 -3062.162,E2 -3062.162} C_VEL
LIN {X 0,Y 558.821,Z 569.98,A -85,B 0,C 180,E1 -3063.605,E2 -3063.605} C_VEL
LIN {X 0,Y 558.788,Z 566.512,A -85,B 0,C 180,E1 -3065.05,E2 -3065.05} C_VEL
LIN {X 0,Y 558.865,Z 561.4,A -85,B 0,C 180,E1 -3066.596,E2 -3066.596} C_VEL
LIN {X 0,Y 558.938,Z 555.605,A -85,B 0,C 180,E1 -3067.95,E2 -3067.95} C_VEL
LIN {X 0,Y 559.004,Z 547.934,A -85,B 0,C 180,E1 -3069.406,E2 -3069.406} C_VEL
LIN {X 0,Y 559.204,Z 539.633,A -85,B 0,C 180,E1 -3070.682,E2 -3070.682} C_VEL
LIN {X 0,Y 559.302,Z 531.262,A -85,B 0,C 180,E1 -3071.782,E2 -3071.782} C_VEL
LIN {X 0,Y 559.536,Z 521.448,A -85,B 0,C 180,E1 -3072.881,E2 -3072.881} C_VEL
LIN {X 0,Y 559.757,Z 510.703,A -85,B 0,C 180,E1 -3073.893,E2 -3073.893} C_VEL
LIN {X 0,Y 560.025,Z 499.232,A -85,B 0,C 180,E1 -3074.82,E2 -3074.82} C_VEL
LIN {X 0,Y 560.269,Z 486.946,A -85,B 0,C 180,E1 -3075.645,E2 -3075.645} C_VEL
LIN {X 0,Y 560.54,Z 475.399,A -85,B 0,C 180,E1 -3076.291,E2 -3076.291} C_VEL
LIN {X 0,Y 560.751,Z 461.339,A -85,B 0,C 180,E1 -3076.941,E2 -3076.941} C_VEL
LIN {X 0,Y 561.009,Z 446.638,A -85,B 0,C 180,E1 -3077.449,E2 -3077.449} C_VEL
LIN {X 0,Y 561.194,Z 433.214,A -85,B 0,C 180,E1 -3077.793,E2 -3077.793} C_VEL
LIN {X 0,Y 561.264,Z 413.889,A -85,B 0,C 180,E1 -3078.103,E2 -3078.103} C_VEL
LIN {X 0,Y 561.442,Z 372.613,A -85,B 0,C 180,E1 -3078.642,E2 -3078.642} C_VEL
LIN {X 0,Y 560.869,Z 366.809,A -85,B 0,C 180,E1 -3078.739,E2 -3078.739} C_VEL
LIN {X 0,Y 555.465,Z 348.178,A -85,B 0,C 180,E1 -3079.172,E2 -3079.172} C_VEL
LIN {X 0,Y 554.838,Z 342.38,A -85,B 0,C 180,E1 -3079.274,E2 -3079.274} C_VEL
LIN {X 0,Y 555.054,Z 273.105,A -85,B 0,C 180,E1 -3080.199,E2 -3080.199} C_VEL
LIN {X 0,Y 553.023,Z 263.785,A -85,B 0,C 180,E1 -3080.424,E2 -3080.424} C_VEL
LIN {X 0,Y 552.975,Z 258.707,A -85,B 0,C 180,E1 -3081.236,E2 -3081.236} C_VEL
LIN {X 0,Y 552.109,Z 254.341,A -85,B 0,C 180,E1 -3082.001,E2 -3082.001} C_VEL
LIN {X 0,Y 552.079,Z 254.338,A -85,B 0,C 180,E1 -3084.839,E2 -3084.839} C_VEL
LIN {X 0,Y 552.097,Z 254.335,A -85,B 0,C 180,E1 -3087.274,E2 -3087.274} C_VEL
LIN {X 0,Y 552.108,Z 254.34,A -85,B 0,C 180,E1 -3090.048,E2 -3090.048} C_VEL
LIN {X 0,Y 552.114,Z 254.331,A -85,B 0,C 180,E1 -3092.845,E2 -3092.845} C_VEL
LIN {X 0,Y 552.069,Z 254.339,A -85,B 0,C 180,E1 -3095.438,E2 -3095.438} C_VEL
LIN {X 0,Y 552.092,Z 254.343,A -85,B 0,C 180,E1 -3097.884,E2 -3097.884} C_VEL
LIN {X 0,Y 552.106,Z 254.333,A -85,B 0,C 180,E1 -3100.48,E2 -3100.48} C_VEL
LIN {X 0,Y 552.105,Z 254.335,A -85,B 0,C 180,E1 -3103.423,E2 -3103.423} C_VEL
LIN {X 0,Y 552.104,Z 254.332,A -85,B 0,C 180,E1 -3106.575,E2 -3106.575} C_VEL
LIN {X 0,Y 552.105,Z 254.337,A -85,B 0,C 180,E1 -3109.518,E2 -3109.518} C_VEL
LIN {X 0,Y 552.089,Z 254.336,A -85,B 0,C 180,E1 -3112.335,E2 -3112.335} C_VEL
LIN {X 0,Y 552.081,Z 254.335,A -85,B 0,C 180,E1 -3115.05,E2 -3115.05} C_VEL
LIN {X 0,Y 552.11,Z 254.34,A -85,B 0,C 180,E1 -3117.68,E2 -3117.68} C_VEL
LIN {X 0,Y 552.106,Z 254.334,A -85,B 0,C 180,E1 -3120.234,E2 -3120.234} C_VEL
LIN {X 0,Y 552.125,Z 254.33,A -85,B 0,C 180,E1 -3123.001,E2 -3123.001} C_VEL
LIN {X 0,Y 552.107,Z 254.334,A -85,B 0,C 180,E1 -3125.16,E2 -3125.16} C_VEL
LIN {X 0,Y 552.12,Z 254.331,A -85,B 0,C 180,E1 -3128.336,E2 -3128.336} C_VEL
LIN {X 0,Y 552.145,Z 254.327,A -85,B 0,C 180,E1 -3130.673,E2 -3130.673} C_VEL
LIN {X 0,Y 552.112,Z 254.339,A -85,B 0,C 180,E1 -3133.736,E2 -3133.736} C_VEL
LIN {X 0,Y 552.125,Z 254.333,A -85,B 0,C 180,E1 -3136.003,E2 -3136.003} C_VEL
LIN {X 0,Y 552.155,Z 254.327,A -85,B 0,C 180,E1 -3138.992,E2 -3138.992} C_VEL
LIN {X 0,Y 552.151,Z 254.33,A -85,B 0,C 180,E1 -3141.951,E2 -3141.951} C_VEL
LIN {X 0,Y 552.22,Z 254.318,A -85,B 0,C 180,E1 -3144.888,E2 -3144.888} C_VEL
LIN {X 0,Y 552.209,Z 254.325,A -85,B 0,C 180,E1 -3147.811,E2 -3147.811} C_VEL
LIN {X 0,Y 552.233,Z 254.316,A -85,B 0,C 180,E1 -3150.728,E2 -3150.728} C_VEL
LIN {X 0,Y 552.196,Z 254.322,A -85,B 0,C 180,E1 -3152.917,E2 -3152.917} C_VEL
LIN {X 0,Y 552.187,Z 254.326,A -85,B 0,C 180,E1 -3155.843,E2 -3155.843} C_VEL
LIN {X 0,Y 552.135,Z 254.329,A -85,B 0,C 180,E1 -3158.785,E2 -3158.785} C_VEL
LIN {X 0,Y 552.152,Z 254.331,A -85,B 0,C 180,E1 -3161.75,E2 -3161.75} C_VEL
LIN {X 0,Y 552.125,Z 254.33,A -85,B 0,C 180,E1 -3164.748,E2 -3164.748} C_VEL
LIN {X 0,Y 552.097,Z 254.337,A -85,B 0,C 180,E1 -3167.788,E2 -3167.788} C_VEL
LIN {X 0,Y 552.118,Z 254.331,A -85,B 0,C 180,E1 -3170.1,E2 -3170.1} C_VEL
LIN {X 0,Y 552.08,Z 254.335,A -85,B 0,C 180,E1 -3172.45,E2 -3172.45} C_VEL
LIN {X 0,Y 552.142,Z 254.336,A -85,B 0,C 180,E1 -3175.35,E2 -3175.35} C_VEL
LIN {X 0,Y 552.106,Z 254.332,A -85,B 0,C 180,E1 -3178.097,E2 -3178.097} C_VEL
LIN {X 0,Y 552.094,Z 254.334,A -85,B 0,C 180,E1 -3180.608,E2 -3180.608} C_VEL
LIN {X 0,Y 552.109,Z 254.338,A -85,B 0,C 180,E1 -3183.185,E2 -3183.185} C_VEL
LIN {X 0,Y 552.09,Z 254.336,A -85,B 0,C 180,E1 -3185.842,E2 -3185.842} C_VEL
LIN {X 0,Y 552.111,Z 254.336,A -85,B 0,C 180,E1 -3189.061,E2 -3189.061} C_VEL
LIN {X 0,Y 552.114,Z 254.338,A -85,B 0,C 180,E1 -3191.445,E2 -3191.445} C_VEL
LIN {X 0,Y 552.082,Z 254.335,A -85,B 0,C 180,E1 -3194.532,E2 -3194.532} C_VEL
LIN {X 0,Y 552.114,Z 254.335,A -85,B 0,C 180,E1 -3197.584,E2 -3197.584} C_VEL
LIN {X 0,Y 552.119,Z 254.33,A -85,B 0,C 180,E1 -3200.473,E2 -3200.473} C_VEL
LIN {X 0,Y 552.096,Z 254.342,A -85,B 0,C 180,E1 -3203.316,E2 -3203.316} C_VEL
LIN {X 0,Y 552.117,Z 254.331,A -85,B 0,C 180,E1 -3205.939,E2 -3205.939} C_VEL
LIN {X 0,Y 552.103,Z 254.333,A -85,B 0,C 180,E1 -3208.541,E2 -3208.541} C_VEL
LIN {X 0,Y 552.109,Z 254.337,A -85,B 0,C 180,E1 -3211.438,E2 -3211.438} C_VEL
LIN {X 0,Y 552.115,Z 254.331,A -85,B 0,C 180,E1 -3214.356,E2 -3214.356} C_VEL
LIN {X 0,Y 552.084,Z 254.338,A -85,B 0,C 180,E1 -3216.758,E2 -3216.758} C_VEL
LIN {X 0,Y 552.112,Z 254.341,A -85,B 0,C 180,E1 -3219.12,E2 -3219.12} C_VEL
LIN {X 0,Y 552.11,Z 254.336,A -85,B 0,C 180,E1 -3221.445,E2 -3221.445} C_VEL
LIN {X 0,Y 552.101,Z 254.334,A -85,B 0,C 180,E1 -3223.738,E2 -3223.738} C_VEL
LIN {X 0,Y 552.119,Z 254.33,A -85,B 0,C 180,E1 -3226.005,E2 -3226.005} C_VEL
LIN {X 0,Y 552.147,Z 254.335,A -85,B 0,C 180,E1 -3228.994,E2 -3228.994} C_VEL
LIN {X 0,Y 552.137,Z 254.328,A -85,B 0,C 180,E1 -3231.952,E2 -3231.952} C_VEL
LIN {X 0,Y 552.213,Z 254.325,A -85,B 0,C 180,E1 -3234.889,E2 -3234.889} C_VEL
LIN {X 0,Y 552.203,Z 254.32,A -85,B 0,C 180,E1 -3237.812,E2 -3237.812} C_VEL
LIN {X 0,Y 552.236,Z 254.321,A -85,B 0,C 180,E1 -3240.73,E2 -3240.73} C_VEL
LIN {X 0,Y 552.197,Z 254.329,A -85,B 0,C 180,E1 -3242.919,E2 -3242.919} C_VEL
LIN {X 0,Y 552.18,Z 254.322,A -85,B 0,C 180,E1 -3245.845,E2 -3245.845} C_VEL
LIN {X 0,Y 552.149,Z 254.333,A -85,B 0,C 180,E1 -3248.786,E2 -3248.786} C_VEL
LIN {X 0,Y 552.151,Z 254.326,A -85,B 0,C 180,E1 -3251.751,E2 -3251.751} C_VEL
LIN {X 0,Y 552.125,Z 254.336,A -85,B 0,C 180,E1 -3254.749,E2 -3254.749} C_VEL
LIN {X 0,Y 552.098,Z 254.333,A -85,B 0,C 180,E1 -3257.789,E2 -3257.789} C_VEL
LIN {X 0,Y 552.119,Z 254.33,A -85,B 0,C 180,E1 -3260.102,E2 -3260.102} C_VEL
LIN {X 0,Y 552.085,Z 254.337,A -85,B 0,C 180,E1 -3262.452,E2 -3262.452} C_VEL
LIN {X 0,Y 552.126,Z 254.332,A -85,B 0,C 180,E1 -3265.347,E2 -3265.347} C_VEL
LIN {X 0,Y 552.098,Z 254.333,A -85,B 0,C 180,E1 -3268.099,E2 -3268.099} C_VEL
LIN {X 0,Y 552.092,Z 254.339,A -85,B 0,C 180,E1 -3270.61,E2 -3270.61} C_VEL
LIN {X 0,Y 552.103,Z 254.336,A -85,B 0,C 180,E1 -3273.187,E2 -3273.187} C_VEL
LIN {X 0,Y 552.076,Z 254.335,A -85,B 0,C 180,E1 -3275.845,E2 -3275.845} C_VEL
LIN {X 0,Y 552.108,Z 254.338,A -85,B 0,C 180,E1 -3278.59,E2 -3278.59} C_VEL
LIN {X 0,Y 552.121,Z 254.331,A -85,B 0,C 180,E1 -3281.446,E2 -3281.446} C_VEL
LIN {X 0,Y 552.083,Z 254.341,A -85,B 0,C 180,E1 -3284.532,E2 -3284.532} C_VEL
LIN {X 0,Y 552.122,Z 254.33,A -85,B 0,C 180,E1 -3287.586,E2 -3287.586} C_VEL
LIN {X 0,Y 552.125,Z 254.336,A -85,B 0,C 180,E1 -3290.474,E2 -3290.474} C_VEL
LIN {X 0,Y 552.092,Z 254.335,A -85,B 0,C 180,E1 -3293.319,E2 -3293.319} C_VEL
LIN {X 0,Y 552.12,Z 254.33,A -85,B 0,C 180,E1 -3295.94,E2 -3295.94} C_VEL
LIN {X 0,Y 552.114,Z 254.338,A -85,B 0,C 180,E1 -3298.542,E2 -3298.542} C_VEL
LIN {X 0,Y 552.109,Z 254.338,A -85,B 0,C 180,E1 -3301.658,E2 -3301.658} C_VEL
LIN {X 0,Y 554.481,Z 264.866,A -85,B 0,C 180,E1 -3303.057,E2 -3303.057} C_VEL
LIN {X 0,Y 554.027,Z 289.623,A -85,B 0,C 180,E1 -3305.972,E2 -3305.972} C_VEL
LIN {X 0,Y 553.531,Z 315.687,A -85,B 0,C 180,E1 -3308.982,E2 -3308.982} C_VEL
LIN {X 0,Y 553.405,Z 321.374,A -85,B 0,C 180,E1 -3309.632,E2 -3309.632} C_VEL
LIN {X 0,Y 555.151,Z 330.466,A -85,B 0,C 180,E1 -3309.816,E2 -3309.816} C_VEL
LIN {X 0,Y 554.486,Z 487.807,A -85,B 0,C 180,E1 -3311.918,E2 -3311.918} C_VEL
LIN {X 0,Y 554.305,Z 503.743,A -85,B 0,C 180,E1 -3312.286,E2 -3312.286} C_VEL
LIN {X 0,Y 554.009,Z 519.063,A -85,B 0,C 180,E1 -3312.8,E2 -3312.8} C_VEL
LIN {X 0,Y 553.781,Z 532.805,A -85,B 0,C 180,E1 -3313.41,E2 -3313.41} C_VEL
LIN {X 0,Y 553.404,Z 546.273,A -85,B 0,C 180,E1 -3314.156,E2 -3314.156} C_VEL
LIN {X 0,Y 553.078,Z 560.146,A -85,B 0,C 180,E1 -3315.103,E2 -3315.103} C_VEL
LIN {X 0,Y 552.759,Z 572.367,A -85,B 0,C 180,E1 -3316.116,E2 -3316.116} C_VEL
LIN {X 0,Y 552.481,Z 584.519,A -85,B 0,C 180,E1 -3317.325,E2 -3317.325} C_VEL
LIN {X 0,Y 552.214,Z 594.493,A -85,B 0,C 180,E1 -3318.514,E2 -3318.514} C_VEL
LIN {X 0,Y 552.124,Z 603.093,A -85,B 0,C 180,E1 -3319.736,E2 -3319.736} C_VEL
LIN {X 0,Y 551.92,Z 610.748,A -85,B 0,C 180,E1 -3321.027,E2 -3321.027} C_VEL
LIN {X 0,Y 551.837,Z 617.095,A -85,B 0,C 180,E1 -3322.316,E2 -3322.316} C_VEL
LIN {X 0,Y 551.758,Z 622.611,A -85,B 0,C 180,E1 -3323.693,E2 -3323.693} C_VEL
LIN {X 0,Y 551.713,Z 626.39,A -85,B 0,C 180,E1 -3324.885,E2 -3324.885} C_VEL
LIN {X 0,Y 551.73,Z 629.89,A -85,B 0,C 180,E1 -3326.349,E2 -3326.349} C_VEL
LIN {X 0,Y 551.654,Z 632.192,A -85,B 0,C 180,E1 -3327.811,E2 -3327.811} C_VEL
LIN {X 0,Y 551.639,Z 633.348,A -85,B 0,C 180,E1 -3329.271,E2 -3329.271} C_VEL
LIN {X 0,Y 551.639,Z 633.347,A -85,B 0,C 180,E1 -3330.731,E2 -3330.731} C_VEL
LIN {X 0,Y 551.654,Z 632.187,A -85,B 0,C 180,E1 -3332.191,E2 -3332.191} C_VEL
LIN {X 0,Y 551.73,Z 629.883,A -85,B 0,C 180,E1 -3333.653,E2 -3333.653} C_VEL
LIN {X 0,Y 551.713,Z 626.384,A -85,B 0,C 180,E1 -3335.117,E2 -3335.117} C_VEL
LIN {X 0,Y 551.782,Z 621.605,A -85,B 0,C 180,E1 -3336.583,E2 -3336.583} C_VEL
LIN {X 0,Y 551.877,Z 615.416,A -85,B 0,C 180,E1 -3338.053,E2 -3338.053} C_VEL
LIN {X 0,Y 551.951,Z 607.639,A -85,B 0,C 180,E1 -3339.529,E2 -3339.529} C_VEL
LIN {X 0,Y 552.185,Z 599.361,A -85,B 0,C 180,E1 -3340.821,E2 -3340.821} C_VEL
LIN {X 0,Y 552.354,Z 589.383,A -85,B 0,C 180,E1 -3342.12,E2 -3342.12} C_VEL
LIN {X 0,Y 552.61,Z 579.177,A -85,B 0,C 180,E1 -3343.234,E2 -3343.234} C_VEL
LIN {X 0,Y 552.91,Z 567.009,A -85,B 0,C 180,E1 -3344.352,E2 -3344.352} C_VEL
LIN {X 0,Y 553.265,Z 554.43,A -85,B 0,C 180,E1 -3345.31,E2 -3345.31} C_VEL
LIN {X 0,Y 553.511,Z 541.491,A -85,B 0,C 180,E1 -3346.127,E2 -3346.127} C_VEL
LIN {X 0,Y 553.84,Z 526.804,A -85,B 0,C 180,E1 -3346.875,E2 -3346.875} C_VEL
LIN {X 0,Y 554.139,Z 512.59,A -85,B 0,C 180,E1 -3347.436,E2 -3347.436} C_VEL
LIN {X 0,Y 554.402,Z 497.478,A -85,B 0,C 180,E1 -3347.876,E2 -3347.876} C_VEL
LIN {X 0,Y 554.508,Z 483.252,A -85,B 0,C 180,E1 -3348.154,E2 -3348.154} C_VEL
LIN {X 0,Y 555.146,Z 330.79,A -85,B 0,C 180,E1 -3350.178,E2 -3350.178} C_VEL
LIN {X 0,Y 553.384,Z 321.161,A -85,B 0,C 180,E1 -3350.374,E2 -3350.374} C_VEL
LIN {X 0,Y 553.742,Z 298.18,A -85,B 0,C 180,E1 -3352.972,E2 -3352.972} C_VEL
LIN {X 0,Y 554.11,Z 275.745,A -85,B 0,C 180,E1 -3355.547,E2 -3355.547} C_VEL
LIN {X 0,Y 554.198,Z 263.619,A -85,B 0,C 180,E1 -3356.96,E2 -3356.96} C_VEL
LIN {X 0,Y 552.14,Z 254.333,A -85,B 0,C 180,E1 -3358.173,E2 -3358.173} C_VEL
LIN {X 0,Y 552.103,Z 254.337,A -85,B 0,C 180,E1 -3360.61,E2 -3360.61} C_VEL
LIN {X 0,Y 552.118,Z 254.341,A -85,B 0,C 180,E1 -3363.186,E2 -3363.186} C_VEL
LIN {X 0,Y 552.09,Z 254.337,A -85,B 0,C 180,E1 -3365.844,E2 -3365.844} C_VEL
LIN {X 0,Y 552.129,Z 254.338,A -85,B 0,C 180,E1 -3369.062,E2 -3369.062} C_VEL
LIN {X 0,Y 552.125,Z 254.334,A -85,B 0,C 180,E1 -3371.446,E2 -3371.446} C_VEL
LIN {X 0,Y 552.096,Z 254.34,A -85,B 0,C 180,E1 -3374.532,E2 -3374.532} C_VEL
LIN {X 0,Y 552.135,Z 254.33,A -85,B 0,C 180,E1 -3377.585,E2 -3377.585} C_VEL
LIN {X 0,Y 552.133,Z 254.336,A -85,B 0,C 180,E1 -3380.473,E2 -3380.473} C_VEL
LIN {X 0,Y 552.104,Z 254.335,A -85,B 0,C 180,E1 -3383.318,E2 -3383.318} C_VEL
LIN {X 0,Y 552.132,Z 254.333,A -85,B 0,C 180,E1 -3385.939,E2 -3385.939} C_VEL
LIN {X 0,Y 552.125,Z 254.339,A -85,B 0,C 180,E1 -3388.541,E2 -3388.541} C_VEL
LIN {X 0,Y 552.103,Z 254.335,A -85,B 0,C 180,E1 -3391.443,E2 -3391.443} C_VEL
LIN {X 0,Y 552.133,Z 254.338,A -85,B 0,C 180,E1 -3394.356,E2 -3394.356} C_VEL
LIN {X 0,Y 552.1,Z 254.34,A -85,B 0,C 180,E1 -3396.758,E2 -3396.758} C_VEL
LIN {X 0,Y 552.138,Z 254.474,A -85,B 0,C 180,E1 -3398.026,E2 -3398.026} C_VEL
LIN {X 0,Y 553.194,Z 259.857,A -85,B 0,C 180,E1 -3398.967,E2 -3398.967} C_VEL
LIN {X 0,Y 553.066,Z 264.317,A -85,B 0,C 180,E1 -3399.686,E2 -3399.686} C_VEL
LIN {X 0,Y 555.121,Z 274.067,A -85,B 0,C 180,E1 -3399.908,E2 -3399.908} C_VEL
LIN {X 0,Y 554.462,Z 427.217,A -85,B 0,C 180,E1 -3401.959,E2 -3401.959} C_VEL
LIN {X 0,Y 554.282,Z 442.814,A -85,B 0,C 180,E1 -3402.307,E2 -3402.307} C_VEL
LIN {X 0,Y 554.041,Z 456.457,A -85,B 0,C 180,E1 -3402.751,E2 -3402.751} C_VEL
LIN {X 0,Y 553.818,Z 469.916,A -85,B 0,C 180,E1 -3403.314,E2 -3403.314} C_VEL
LIN {X 0,Y 553.47,Z 483.855,A -85,B 0,C 180,E1 -3404.062,E2 -3404.062} C_VEL
LIN {X 0,Y 553.186,Z 495.997,A -85,B 0,C 180,E1 -3404.848,E2 -3404.848} C_VEL
LIN {X 0,Y 552.869,Z 508.615,A -85,B 0,C 180,E1 -3405.835,E2 -3405.835} C_VEL
LIN {X 0,Y 552.61,Z 518.657,A -85,B 0,C 180,E1 -3406.766,E2 -3406.766} C_VEL
LIN {X 0,Y 552.362,Z 529.001,A -85,B 0,C 180,E1 -3407.881,E2 -3407.881} C_VEL
LIN {X 0,Y 552.176,Z 538.984,A -85,B 0,C 180,E1 -3409.179,E2 -3409.179} C_VEL
LIN {X 0,Y 552.009,Z 546.237,A -85,B 0,C 180,E1 -3410.288,E2 -3410.288} C_VEL
LIN {X 0,Y 551.905,Z 553.414,A -85,B 0,C 180,E1 -3411.579,E2 -3411.579} C_VEL
LIN {X 0,Y 551.816,Z 559.981,A -85,B 0,C 180,E1 -3413.05,E2 -3413.05} C_VEL
LIN {X 0,Y 551.785,Z 565.199,A -85,B 0,C 180,E1 -3414.518,E2 -3414.518} C_VEL
LIN {X 0,Y 551.705,Z 568.203,A -85,B 0,C 180,E1 -3415.616,E2 -3415.616} C_VEL
LIN {X 0,Y 551.718,Z 571.103,A -85,B 0,C 180,E1 -3417.079,E2 -3417.079} C_VEL
LIN {X 0,Y 551.643,Z 572.85,A -85,B 0,C 180,E1 -3418.539,E2 -3418.539} C_VEL
LIN {X 0,Y 551.637,Z 573.496,A -85,B 0,C 180,E1 -3419.999,E2 -3419.999} C_VEL
LIN {X 0,Y 551.642,Z 572.932,A -85,B 0,C 180,E1 -3421.459,E2 -3421.459} C_VEL
LIN {X 0,Y 551.72,Z 571.24,A -85,B 0,C 180,E1 -3422.92,E2 -3422.92} C_VEL
LIN {X 0,Y 551.706,Z 568.426,A -85,B 0,C 180,E1 -3424.383,E2 -3424.383} C_VEL
LIN {X 0,Y 551.789,Z 564.284,A -85,B 0,C 180,E1 -3425.848,E2 -3425.848} C_VEL
LIN {X 0,Y 551.819,Z 558.881,A -85,B 0,C 180,E1 -3427.316,E2 -3427.316} C_VEL
LIN {X 0,Y 551.909,Z 551.957,A -85,B 0,C 180,E1 -3428.789,E2 -3428.789} C_VEL
LIN {X 0,Y 552.068,Z 544.524,A -85,B 0,C 180,E1 -3430.08,E2 -3430.08} C_VEL
LIN {X 0,Y 552.231,Z 534.742,A -85,B 0,C 180,E1 -3431.492,E2 -3431.492} C_VEL
LIN {X 0,Y 552.417,Z 526.509,A -85,B 0,C 180,E1 -3432.49,E2 -3432.49} C_VEL
LIN {X 0,Y 552.674,Z 515.817,A -85,B 0,C 180,E1 -3433.606,E2 -3433.606} C_VEL
LIN {X 0,Y 552.994,Z 504.08,A -85,B 0,C 180,E1 -3434.63,E2 -3434.63} C_VEL
LIN {X 0,Y 553.267,Z 492.659,A -85,B 0,C 180,E1 -3435.471,E2 -3435.471} C_VEL
LIN {X 0,Y 553.604,Z 478.996,A -85,B 0,C 180,E1 -3436.312,E2 -3436.312} C_VEL
LIN {X 0,Y 553.882,Z 465.592,A -85,B 0,C 180,E1 -3436.967,E2 -3436.967} C_VEL
LIN {X 0,Y 554.151,Z 452.515,A -85,B 0,C 180,E1 -3437.482,E2 -3437.482} C_VEL
LIN {X 0,Y 554.328,Z 437.387,A -85,B 0,C 180,E1 -3437.921,E2 -3437.921} C_VEL
LIN {X 0,Y 554.468,Z 424.115,A -85,B 0,C 180,E1 -3438.182,E2 -3438.182} C_VEL
LIN {X 0,Y 554.838,Z 342.38,A -85,B 0,C 180,E1 -3439.274,E2 -3439.274} C_VEL
LIN {X 0,Y 554.23,Z 336.584,A -85,B 0,C 180,E1 -3439.377,E2 -3439.377} C_VEL
LIN {X 0,Y 548.901,Z 317.951,A -85,B 0,C 180,E1 -3439.82,E2 -3439.82} C_VEL
LIN {X 0,Y 548.32,Z 312.15,A -85,B 0,C 180,E1 -3439.92,E2 -3439.92} C_VEL
LIN {X 0,Y 548.338,Z 273.991,A -85,B 0,C 180,E1 -3440.445,E2 -3440.445} C_VEL
LIN {X 0,Y 546.142,Z 264.073,A -85,B 0,C 180,E1 -3440.689,E2 -3440.689} C_VEL
LIN {X 0,Y 545.85,Z 259.055,A -85,B 0,C 180,E1 -3441.509,E2 -3441.509} C_VEL
LIN {X 0,Y 545.069,Z 255.218,A -85,B 0,C 180,E1 -3442.181,E2 -3442.181} C_VEL
LIN {X 0,Y 545.064,Z 255.212,A -85,B 0,C 180,E1 -3445.181,E2 -3445.181} C_VEL
LIN {X 0,Y 545.057,Z 255.216,A -85,B 0,C 180,E1 -3447.657,E2 -3447.657} C_VEL
LIN {X 0,Y 545.054,Z 255.215,A -85,B 0,C 180,E1 -3450.241,E2 -3450.241} C_VEL
LIN {X 0,Y 545.078,Z 255.207,A -85,B 0,C 180,E1 -3453.061,E2 -3453.061} C_VEL
LIN {X 0,Y 545.024,Z 255.22,A -85,B 0,C 180,E1 -3455.671,E2 -3455.671} C_VEL
LIN {X 0,Y 545.048,Z 255.215,A -85,B 0,C 180,E1 -3458.237,E2 -3458.237} C_VEL
LIN {X 0,Y 545.078,Z 255.208,A -85,B 0,C 180,E1 -3460.472,E2 -3460.472} C_VEL
LIN {X 0,Y 545.048,Z 255.211,A -85,B 0,C 180,E1 -3463.108,E2 -3463.108} C_VEL
LIN {X 0,Y 545.047,Z 255.214,A -85,B 0,C 180,E1 -3466.225,E2 -3466.225} C_VEL
LIN {X 0,Y 545.079,Z 255.207,A -85,B 0,C 180,E1 -3468.884,E2 -3468.884} C_VEL
LIN {X 0,Y 545.049,Z 255.22,A -85,B 0,C 180,E1 -3471.762,E2 -3471.762} C_VEL
LIN {X 0,Y 545.034,Z 255.213,A -85,B 0,C 180,E1 -3474.531,E2 -3474.531} C_VEL
LIN {X 0,Y 545.061,Z 255.211,A -85,B 0,C 180,E1 -3477.21,E2 -3477.21} C_VEL
LIN {X 0,Y 545.059,Z 255.218,A -85,B 0,C 180,E1 -3479.809,E2 -3479.809} C_VEL
LIN {X 0,Y 545.055,Z 255.211,A -85,B 0,C 180,E1 -3482.342,E2 -3482.342} C_VEL
LIN {X 0,Y 545.1,Z 255.204,A -85,B 0,C 180,E1 -3484.819,E2 -3484.819} C_VEL
LIN {X 0,Y 545.03,Z 255.216,A -85,B 0,C 180,E1 -3487.241,E2 -3487.241} C_VEL
LIN {X 0,Y 545.11,Z 255.204,A -85,B 0,C 180,E1 -3490.414,E2 -3490.414} C_VEL
LIN {X 0,Y 545.069,Z 255.216,A -85,B 0,C 180,E1 -3493.52,E2 -3493.52} C_VEL
LIN {X 0,Y 545.085,Z 255.213,A -85,B 0,C 180,E1 -3495.819,E2 -3495.819} C_VEL
LIN {X 0,Y 545.111,Z 255.203,A -85,B 0,C 180,E1 -3498.848,E2 -3498.848} C_VEL
LIN {X 0,Y 545.121,Z 255.207,A -85,B 0,C 180,E1 -3501.846,E2 -3501.846} C_VEL
LIN {X 0,Y 545.196,Z 255.193,A -85,B 0,C 180,E1 -3504.822,E2 -3504.822} C_VEL
LIN {X 0,Y 545.182,Z 255.2,A -85,B 0,C 180,E1 -3507.783,E2 -3507.783} C_VEL
LIN {X 0,Y 545.203,Z 255.192,A -85,B 0,C 180,E1 -3510.738,E2 -3510.738} C_VEL
LIN {X 0,Y 545.163,Z 255.198,A -85,B 0,C 180,E1 -3512.955,E2 -3512.955} C_VEL
LIN {X 0,Y 545.158,Z 255.201,A -85,B 0,C 180,E1 -3515.919,E2 -3515.919} C_VEL
LIN {X 0,Y 545.098,Z 255.206,A -85,B 0,C 180,E1 -3518.899,E2 -3518.899} C_VEL
LIN {X 0,Y 545.124,Z 255.205,A -85,B 0,C 180,E1 -3521.903,E2 -3521.903} C_VEL
LIN {X 0,Y 545.074,Z 255.21,A -85,B 0,C 180,E1 -3524.943,E2 -3524.943} C_VEL
LIN {X 0,Y 545.066,Z 255.21,A -85,B 0,C 180,E1 -3528.025,E2 -3528.025} C_VEL
LIN {X 0,Y 545.083,Z 255.206,A -85,B 0,C 180,E1 -3530.371,E2 -3530.371} C_VEL
LIN {X 0,Y 545.068,Z 255.216,A -85,B 0,C 180,E1 -3533.559,E2 -3533.559} C_VEL
LIN {X 0,Y 545.066,Z 255.21,A -85,B 0,C 180,E1 -3536,E2 -3536} C_VEL
LIN {X 0,Y 545.075,Z 255.209,A -85,B 0,C 180,E1 -3538.747,E2 -3538.747} C_VEL
LIN {X 0,Y 545.064,Z 255.213,A -85,B 0,C 180,E1 -3541.682,E2 -3541.682} C_VEL
LIN {X 0,Y 545.067,Z 255.209,A -85,B 0,C 180,E1 -3544.562,E2 -3544.562} C_VEL
LIN {X 0,Y 545.024,Z 255.223,A -85,B 0,C 180,E1 -3547.303,E2 -3547.303} C_VEL
LIN {X 0,Y 545.059,Z 255.21,A -85,B 0,C 180,E1 -3550.141,E2 -3550.141} C_VEL
LIN {X 0,Y 545.071,Z 255.214,A -85,B 0,C 180,E1 -3553.105,E2 -3553.105} C_VEL
LIN {X 0,Y 545.05,Z 255.211,A -85,B 0,C 180,E1 -3556.224,E2 -3556.224} C_VEL
LIN {X 0,Y 545.076,Z 255.211,A -85,B 0,C 180,E1 -3558.886,E2 -3558.886} C_VEL
LIN {X 0,Y 545.038,Z 255.214,A -85,B 0,C 180,E1 -3561.763,E2 -3561.763} C_VEL
LIN {X 0,Y 545.042,Z 255.212,A -85,B 0,C 180,E1 -3564.533,E2 -3564.533} C_VEL
LIN {X 0,Y 545.066,Z 255.219,A -85,B 0,C 180,E1 -3567.212,E2 -3567.212} C_VEL
LIN {X 0,Y 545.051,Z 255.212,A -85,B 0,C 180,E1 -3569.811,E2 -3569.811} C_VEL
LIN {X 0,Y 545.074,Z 255.208,A -85,B 0,C 180,E1 -3572.344,E2 -3572.344} C_VEL
LIN {X 0,Y 545.102,Z 255.208,A -85,B 0,C 180,E1 -3574.821,E2 -3574.821} C_VEL
LIN {X 0,Y 545.024,Z 255.222,A -85,B 0,C 180,E1 -3577.243,E2 -3577.243} C_VEL
LIN {X 0,Y 545.106,Z 255.204,A -85,B 0,C 180,E1 -3580.415,E2 -3580.415} C_VEL
LIN {X 0,Y 545.057,Z 255.213,A -85,B 0,C 180,E1 -3583.521,E2 -3583.521} C_VEL
LIN {X 0,Y 545.079,Z 255.208,A -85,B 0,C 180,E1 -3585.82,E2 -3585.82} C_VEL
LIN {X 0,Y 545.103,Z 255.21,A -85,B 0,C 180,E1 -3588.85,E2 -3588.85} C_VEL
LIN {X 0,Y 545.108,Z 255.204,A -85,B 0,C 180,E1 -3591.847,E2 -3591.847} C_VEL
LIN {X 0,Y 545.189,Z 255.199,A -85,B 0,C 180,E1 -3594.823,E2 -3594.823} C_VEL
LIN {X 0,Y 545.176,Z 255.195,A -85,B 0,C 180,E1 -3597.784,E2 -3597.784} C_VEL
LIN {X 0,Y 545.205,Z 255.196,A -85,B 0,C 180,E1 -3600.739,E2 -3600.739} C_VEL
LIN {X 0,Y 545.163,Z 255.206,A -85,B 0,C 180,E1 -3602.956,E2 -3602.956} C_VEL
LIN {X 0,Y 545.152,Z 255.198,A -85,B 0,C 180,E1 -3605.92,E2 -3605.92} C_VEL
LIN {X 0,Y 545.108,Z 255.212,A -85,B 0,C 180,E1 -3608.901,E2 -3608.901} C_VEL
LIN {X 0,Y 545.123,Z 255.201,A -85,B 0,C 180,E1 -3611.905,E2 -3611.905} C_VEL
LIN {X 0,Y 545.074,Z 255.217,A -85,B 0,C 180,E1 -3614.944,E2 -3614.944} C_VEL
LIN {X 0,Y 545.066,Z 255.209,A -85,B 0,C 180,E1 -3618.027,E2 -3618.027} C_VEL
LIN {X 0,Y 545.085,Z 255.208,A -85,B 0,C 180,E1 -3620.373,E2 -3620.373} C_VEL
LIN {X 0,Y 545.07,Z 255.209,A -85,B 0,C 180,E1 -3623.56,E2 -3623.56} C_VEL
LIN {X 0,Y 545.066,Z 255.209,A -85,B 0,C 180,E1 -3626.002,E2 -3626.002} C_VEL
LIN {X 0,Y 545.079,Z 255.215,A -85,B 0,C 180,E1 -3628.749,E2 -3628.749} C_VEL
LIN {X 0,Y 545.047,Z 255.211,A -85,B 0,C 180,E1 -3631.68,E2 -3631.68} C_VEL
LIN {X 0,Y 545.062,Z 255.215,A -85,B 0,C 180,E1 -3634.565,E2 -3634.565} C_VEL
LIN {X 0,Y 545.026,Z 255.216,A -85,B 0,C 180,E1 -3637.305,E2 -3637.305} C_VEL
LIN {X 0,Y 545.056,Z 255.211,A -85,B 0,C 180,E1 -3640.144,E2 -3640.144} C_VEL
LIN {X 0,Y 545.07,Z 255.212,A -85,B 0,C 180,E1 -3643.108,E2 -3643.108} C_VEL
LIN {X 0,Y 545.042,Z 255.214,A -85,B 0,C 180,E1 -3646.227,E2 -3646.227} C_VEL
LIN {X 0,Y 545.074,Z 255.216,A -85,B 0,C 180,E1 -3648.887,E2 -3648.887} C_VEL
LIN {X 0,Y 545.076,Z 255.216,A -85,B 0,C 180,E1 -3650.82,E2 -3650.82} C_VEL
LIN {X 0,Y 545.028,Z 255.214,A -85,B 0,C 180,E1 -3653.62,E2 -3653.62} C_VEL
LIN {X 0,Y 545.059,Z 255.214,A -85,B 0,C 180,E1 -3656.329,E2 -3656.329} C_VEL
LIN {X 0,Y 545.06,Z 255.217,A -85,B 0,C 180,E1 -3658.953,E2 -3658.953} C_VEL
LIN {X 0,Y 545.089,Z 255.329,A -85,B 0,C 180,E1 -3661.42,E2 -3661.42} C_VEL
LIN {X 0,Y 547.657,Z 266.274,A -85,B 0,C 180,E1 -3662.9,E2 -3662.9} C_VEL
LIN {X 0,Y 547.245,Z 288.329,A -85,B 0,C 180,E1 -3665.534,E2 -3665.534} C_VEL
LIN {X 0,Y 546.681,Z 315.407,A -85,B 0,C 180,E1 -3668.706,E2 -3668.706} C_VEL
LIN {X 0,Y 546.565,Z 321.214,A -85,B 0,C 180,E1 -3669.373,E2 -3669.373} C_VEL
LIN {X 0,Y 548.43,Z 332.022,A -85,B 0,C 180,E1 -3669.597,E2 -3669.597} C_VEL
LIN {X 0,Y 547.7,Z 487.84,A -85,B 0,C 180,E1 -3671.7,E2 -3671.7} C_VEL
LIN {X 0,Y 547.525,Z 503.384,A -85,B 0,C 180,E1 -3672.059,E2 -3672.059} C_VEL
LIN {X 0,Y 547.217,Z 518.949,A -85,B 0,C 180,E1 -3672.579,E2 -3672.579} C_VEL
LIN {X 0,Y 546.938,Z 532.808,A -85,B 0,C 180,E1 -3673.196,E2 -3673.196} C_VEL
LIN {X 0,Y 546.528,Z 546.273,A -85,B 0,C 180,E1 -3673.951,E2 -3673.951} C_VEL
LIN {X 0,Y 546.149,Z 560.148,A -85,B 0,C 180,E1 -3674.91,E2 -3674.91} C_VEL
LIN {X 0,Y 545.816,Z 572.369,A -85,B 0,C 180,E1 -3675.935,E2 -3675.935} C_VEL
LIN {X 0,Y 545.51,Z 584.519,A -85,B 0,C 180,E1 -3677.161,E2 -3677.161} C_VEL
LIN {X 0,Y 545.174,Z 595.113,A -85,B 0,C 180,E1 -3678.447,E2 -3678.447} C_VEL
LIN {X 0,Y 545.049,Z 604.303,A -85,B 0,C 180,E1 -3679.789,E2 -3679.789} C_VEL
LIN {X 0,Y 544.845,Z 611.756,A -85,B 0,C 180,E1 -3681.097,E2 -3681.097} C_VEL
LIN {X 0,Y 544.744,Z 618.705,A -85,B 0,C 180,E1 -3682.588,E2 -3682.588} C_VEL
LIN {X 0,Y 544.706,Z 624.166,A -85,B 0,C 180,E1 -3684.077,E2 -3684.077} C_VEL
LIN {X 0,Y 544.605,Z 628.294,A -85,B 0,C 180,E1 -3685.56,E2 -3685.56} C_VEL
LIN {X 0,Y 544.644,Z 631.186,A -85,B 0,C 180,E1 -3687.042,E2 -3687.042} C_VEL
LIN {X 0,Y 544.543,Z 632.91,A -85,B 0,C 180,E1 -3688.522,E2 -3688.522} C_VEL
LIN {X 0,Y 544.538,Z 633.5,A -85,B 0,C 180,E1 -3690.001,E2 -3690.001} C_VEL
LIN {X 0,Y 544.543,Z 632.907,A -85,B 0,C 180,E1 -3691.48,E2 -3691.48} C_VEL
LIN {X 0,Y 544.644,Z 631.179,A -85,B 0,C 180,E1 -3692.96,E2 -3692.96} C_VEL
LIN {X 0,Y 544.605,Z 628.286,A -85,B 0,C 180,E1 -3694.442,E2 -3694.442} C_VEL
LIN {X 0,Y 544.702,Z 624.162,A -85,B 0,C 180,E1 -3695.926,E2 -3695.926} C_VEL
LIN {X 0,Y 544.746,Z 618.697,A -85,B 0,C 180,E1 -3697.414,E2 -3697.414} C_VEL
LIN {X 0,Y 544.846,Z 611.739,A -85,B 0,C 180,E1 -3698.905,E2 -3698.905} C_VEL
LIN {X 0,Y 545.074,Z 603.076,A -85,B 0,C 180,E1 -3700.4,E2 -3700.4} C_VEL
LIN {X 0,Y 545.239,Z 593.7,A -85,B 0,C 180,E1 -3701.735,E2 -3701.735} C_VEL
LIN {X 0,Y 545.509,Z 584.5,A -85,B 0,C 180,E1 -3702.841,E2 -3702.841} C_VEL
LIN {X 0,Y 545.792,Z 572.35,A -85,B 0,C 180,E1 -3704.067,E2 -3704.067} C_VEL
LIN {X 0,Y 546.195,Z 559.798,A -85,B 0,C 180,E1 -3705.116,E2 -3705.116} C_VEL
LIN {X 0,Y 546.532,Z 546.236,A -85,B 0,C 180,E1 -3706.051,E2 -3706.051} C_VEL
LIN {X 0,Y 546.974,Z 532.757,A -85,B 0,C 180,E1 -3706.805,E2 -3706.805} C_VEL
LIN {X 0,Y 547.233,Z 518.908,A -85,B 0,C 180,E1 -3707.422,E2 -3707.422} C_VEL
LIN {X 0,Y 547.482,Z 504.025,A -85,B 0,C 180,E1 -3707.921,E2 -3707.921} C_VEL
LIN {X 0,Y 547.67,Z 488.169,A -85,B 0,C 180,E1 -3708.29,E2 -3708.29} C_VEL
LIN {X 0,Y 548.413,Z 332.124,A -85,B 0,C 180,E1 -3710.394,E2 -3710.394} C_VEL
LIN {X 0,Y 546.484,Z 320.609,A -85,B 0,C 180,E1 -3710.636,E2 -3710.636} C_VEL
LIN {X 0,Y 546.91,Z 294.281,A -85,B 0,C 180,E1 -3713.658,E2 -3713.658} C_VEL
LIN {X 0,Y 547.364,Z 269.959,A -85,B 0,C 180,E1 -3716.499,E2 -3716.499} C_VEL
LIN {X 0,Y 547.301,Z 264.925,A -85,B 0,C 180,E1 -3717.103,E2 -3717.103} C_VEL
LIN {X 0,Y 545.059,Z 255.216,A -85,B 0,C 180,E1 -3718.391,E2 -3718.391} C_VEL
LIN {X 0,Y 545.069,Z 255.217,A -85,B 0,C 180,E1 -3721.048,E2 -3721.048} C_VEL
LIN {X 0,Y 545.069,Z 255.214,A -85,B 0,C 180,E1 -3723.672,E2 -3723.672} C_VEL
LIN {X 0,Y 545.075,Z 255.217,A -85,B 0,C 180,E1 -3726.926,E2 -3726.926} C_VEL
LIN {X 0,Y 545.073,Z 255.211,A -85,B 0,C 180,E1 -3730.143,E2 -3730.143} C_VEL
LIN {X 0,Y 545.084,Z 255.215,A -85,B 0,C 180,E1 -3733.107,E2 -3733.107} C_VEL
LIN {X 0,Y 545.061,Z 255.213,A -85,B 0,C 180,E1 -3736.226,E2 -3736.226} C_VEL
LIN {X 0,Y 545.087,Z 255.214,A -85,B 0,C 180,E1 -3738.886,E2 -3738.886} C_VEL
LIN {X 0,Y 545.084,Z 255.215,A -85,B 0,C 180,E1 -3740.818,E2 -3740.818} C_VEL
LIN {X 0,Y 545.04,Z 255.214,A -85,B 0,C 180,E1 -3743.619,E2 -3743.619} C_VEL
LIN {X 0,Y 545.071,Z 255.217,A -85,B 0,C 180,E1 -3746.328,E2 -3746.328} C_VEL
LIN {X 0,Y 545.071,Z 255.213,A -85,B 0,C 180,E1 -3748.952,E2 -3748.952} C_VEL
LIN {X 0,Y 545.081,Z 255.21,A -85,B 0,C 180,E1 -3751.506,E2 -3751.506} C_VEL
LIN {X 0,Y 545.092,Z 255.214,A -85,B 0,C 180,E1 -3754.493,E2 -3754.493} C_VEL
LIN {X 0,Y 545.04,Z 255.218,A -85,B 0,C 180,E1 -3757.242,E2 -3757.242} C_VEL
LIN {X 0,Y 545.084,Z 255.288,A -85,B 0,C 180,E1 -3757.769,E2 -3757.769} C_VEL
LIN {X 0,Y 546.378,Z 261.628,A -85,B 0,C 180,E1 -3758.89,E2 -3758.89} C_VEL
LIN {X 0,Y 546.242,Z 264.891,A -85,B 0,C 180,E1 -3759.42,E2 -3759.42} C_VEL
LIN {X 0,Y 548.456,Z 274.658,A -85,B 0,C 180,E1 -3759.66,E2 -3759.66} C_VEL
LIN {X 0,Y 547.653,Z 428.487,A -85,B 0,C 180,E1 -3761.776,E2 -3761.776} C_VEL
LIN {X 0,Y 547.455,Z 444.506,A -85,B 0,C 180,E1 -3762.151,E2 -3762.151} C_VEL
LIN {X 0,Y 547.194,Z 458.613,A -85,B 0,C 180,E1 -3762.625,E2 -3762.625} C_VEL
LIN {X 0,Y 546.865,Z 473.507,A -85,B 0,C 180,E1 -3763.288,E2 -3763.288} C_VEL
LIN {X 0,Y 546.59,Z 485.377,A -85,B 0,C 180,E1 -3763.951,E2 -3763.951} C_VEL
LIN {X 0,Y 546.233,Z 497.987,A -85,B 0,C 180,E1 -3764.792,E2 -3764.792} C_VEL
LIN {X 0,Y 545.907,Z 509.673,A -85,B 0,C 180,E1 -3765.746,E2 -3765.746} C_VEL
LIN {X 0,Y 545.644,Z 518.654,A -85,B 0,C 180,E1 -3766.594,E2 -3766.594} C_VEL
LIN {X 0,Y 545.363,Z 529.006,A -85,B 0,C 180,E1 -3767.723,E2 -3767.723} C_VEL
LIN {X 0,Y 545.139,Z 537.685,A -85,B 0,C 180,E1 -3768.849,E2 -3768.849} C_VEL
LIN {X 0,Y 544.984,Z 545.097,A -85,B 0,C 180,E1 -3769.974,E2 -3769.974} C_VEL
LIN {X 0,Y 544.851,Z 551.458,A -85,B 0,C 180,E1 -3771.095,E2 -3771.095} C_VEL
LIN {X 0,Y 544.746,Z 558.519,A -85,B 0,C 180,E1 -3772.587,E2 -3772.587} C_VEL
LIN {X 0,Y 544.708,Z 563.983,A -85,B 0,C 180,E1 -3774.075,E2 -3774.075} C_VEL
LIN {X 0,Y 544.605,Z 568.208,A -85,B 0,C 180,E1 -3775.559,E2 -3775.559} C_VEL
LIN {X 0,Y 544.645,Z 571.099,A -85,B 0,C 180,E1 -3777.041,E2 -3777.041} C_VEL
LIN {X 0,Y 544.544,Z 572.845,A -85,B 0,C 180,E1 -3778.52,E2 -3778.52} C_VEL
LIN {X 0,Y 544.537,Z 573.496,A -85,B 0,C 180,E1 -3779.999,E2 -3779.999} C_VEL
LIN {X 0,Y 544.544,Z 572.926,A -85,B 0,C 180,E1 -3781.479,E2 -3781.479} C_VEL
LIN {X 0,Y 544.646,Z 571.235,A -85,B 0,C 180,E1 -3782.958,E2 -3782.958} C_VEL
LIN {X 0,Y 544.606,Z 568.428,A -85,B 0,C 180,E1 -3784.44,E2 -3784.44} C_VEL
LIN {X 0,Y 544.702,Z 564.278,A -85,B 0,C 180,E1 -3785.924,E2 -3785.924} C_VEL
LIN {X 0,Y 544.727,Z 560.333,A -85,B 0,C 180,E1 -3787.04,E2 -3787.04} C_VEL
LIN {X 0,Y 544.818,Z 553.867,A -85,B 0,C 180,E1 -3788.53,E2 -3788.53} C_VEL
LIN {X 0,Y 544.979,Z 545.655,A -85,B 0,C 180,E1 -3790.025,E2 -3790.025} C_VEL
LIN {X 0,Y 545.098,Z 538.311,A -85,B 0,C 180,E1 -3791.15,E2 -3791.15} C_VEL
LIN {X 0,Y 545.37,Z 528.158,A -85,B 0,C 180,E1 -3792.465,E2 -3792.465} C_VEL
LIN {X 0,Y 545.675,Z 517.678,A -85,B 0,C 180,E1 -3793.594,E2 -3793.594} C_VEL
LIN {X 0,Y 545.986,Z 506.429,A -85,B 0,C 180,E1 -3794.632,E2 -3794.632} C_VEL
LIN {X 0,Y 546.358,Z 493.802,A -85,B 0,C 180,E1 -3795.59,E2 -3795.59} C_VEL
LIN {X 0,Y 546.649,Z 482.188,A -85,B 0,C 180,E1 -3796.333,E2 -3796.333} C_VEL
LIN {X 0,Y 547.037,Z 467.549,A -85,B 0,C 180,E1 -3797.09,E2 -3797.09} C_VEL
LIN {X 0,Y 547.286,Z 454.755,A -85,B 0,C 180,E1 -3797.612,E2 -3797.612} C_VEL
LIN {X 0,Y 547.533,Z 439.899,A -85,B 0,C 180,E1 -3798.075,E2 -3798.075} C_VEL
LIN {X 0,Y 547.68,Z 425.805,A -85,B 0,C 180,E1 -3798.368,E2 -3798.368} C_VEL
LIN {X 0,Y 548.32,Z 312.15,A -85,B 0,C 180,E1 -3799.92,E2 -3799.92} C_VEL
LIN {X 0,Y 547.735,Z 306.349,A -85,B 0,C 180,E1 -3800.022,E2 -3800.022} C_VEL
LIN {X 0,Y 542.376,Z 287.744,A -85,B 0,C 180,E1 -3800.481,E2 -3800.481} C_VEL
LIN {X 0,Y 541.778,Z 281.95,A -85,B 0,C 180,E1 -3800.585,E2 -3800.585} C_VEL
LIN {X 0,Y 541.714,Z 275.155,A -85,B 0,C 180,E1 -3800.69,E2 -3800.69} C_VEL
LIN {X 0,Y 539.261,Z 264.293,A -85,B 0,C 180,E1 -3800.973,E2 -3800.973} C_VEL
LIN {X 0,Y 538.766,Z 259.786,A -85,B 0,C 180,E1 -3801.731,E2 -3801.731} C_VEL
LIN {X 0,Y 538.018,Z 256.096,A -85,B 0,C 180,E1 -3802.386,E2 -3802.386} C_VEL
LIN {X 0,Y 538.03,Z 256.092,A -85,B 0,C 180,E1 -3805.534,E2 -3805.534} C_VEL
LIN {X 0,Y 538.02,Z 256.095,A -85,B 0,C 180,E1 -3808.05,E2 -3808.05} C_VEL
LIN {X 0,Y 538.011,Z 256.089,A -85,B 0,C 180,E1 -3810.626,E2 -3810.626} C_VEL
LIN {X 0,Y 538.046,Z 256.085,A -85,B 0,C 180,E1 -3813.282,E2 -3813.282} C_VEL
LIN {X 0,Y 537.988,Z 256.098,A -85,B 0,C 180,E1 -3816.004,E2 -3816.004} C_VEL
LIN {X 0,Y 538.01,Z 256.088,A -85,B 0,C 180,E1 -3818.83,E2 -3818.83} C_VEL
LIN {X 0,Y 538.028,Z 256.094,A -85,B 0,C 180,E1 -3821.772,E2 -3821.772} C_VEL
LIN {X 0,Y 538.004,Z 256.088,A -85,B 0,C 180,E1 -3824.861,E2 -3824.861} C_VEL
LIN {X 0,Y 538.026,Z 256.09,A -85,B 0,C 180,E1 -3828.12,E2 -3828.12} C_VEL
LIN {X 0,Y 538.029,Z 256.087,A -85,B 0,C 180,E1 -3830.414,E2 -3830.414} C_VEL
LIN {X 0,Y 538.02,Z 256.087,A -85,B 0,C 180,E1 -3833.066,E2 -3833.066} C_VEL
LIN {X 0,Y 538.011,Z 256.096,A -85,B 0,C 180,E1 -3835.825,E2 -3835.825} C_VEL
LIN {X 0,Y 538.004,Z 256.089,A -85,B 0,C 180,E1 -3838.498,E2 -3838.498} C_VEL
LIN {X 0,Y 538.016,Z 256.088,A -85,B 0,C 180,E1 -3841.096,E2 -3841.096} C_VEL
LIN {X 0,Y 538.031,Z 256.093,A -85,B 0,C 180,E1 -3843.632,E2 -3843.632} C_VEL
LIN {X 0,Y 538.001,Z 256.092,A -85,B 0,C 180,E1 -3846.121,E2 -3846.121} C_VEL
LIN {X 0,Y 538.032,Z 256.089,A -85,B 0,C 180,E1 -3849.347,E2 -3849.347} C_VEL
LIN {X 0,Y 538.029,Z 256.085,A -85,B 0,C 180,E1 -3852.467,E2 -3852.467} C_VEL
LIN {X 0,Y 538.055,Z 256.092,A -85,B 0,C 180,E1 -3855.63,E2 -3855.63} C_VEL
LIN {X 0,Y 538.07,Z 256.08,A -85,B 0,C 180,E1 -3858.7,E2 -3858.7} C_VEL
LIN {X 0,Y 538.078,Z 256.087,A -85,B 0,C 180,E1 -3861.739,E2 -3861.739} C_VEL
LIN {X 0,Y 538.153,Z 256.07,A -85,B 0,C 180,E1 -3864.754,E2 -3864.754} C_VEL
LIN {X 0,Y 538.154,Z 256.076,A -85,B 0,C 180,E1 -3867.754,E2 -3867.754} C_VEL
LIN {X 0,Y 538.173,Z 256.068,A -85,B 0,C 180,E1 -3870.747,E2 -3870.747} C_VEL
LIN {X 0,Y 538.129,Z 256.075,A -85,B 0,C 180,E1 -3872.993,E2 -3872.993} C_VEL
LIN {X 0,Y 538.109,Z 256.078,A -85,B 0,C 180,E1 -3875.996,E2 -3875.996} C_VEL
LIN {X 0,Y 538.051,Z 256.085,A -85,B 0,C 180,E1 -3879.017,E2 -3879.017} C_VEL
LIN {X 0,Y 538.072,Z 256.082,A -85,B 0,C 180,E1 -3882.062,E2 -3882.062} C_VEL
LIN {X 0,Y 538.034,Z 256.089,A -85,B 0,C 180,E1 -3885.143,E2 -3885.143} C_VEL
LIN {X 0,Y 538.018,Z 256.087,A -85,B 0,C 180,E1 -3888.269,E2 -3888.269} C_VEL
LIN {X 0,Y 538.027,Z 256.086,A -85,B 0,C 180,E1 -3890.651,E2 -3890.651} C_VEL
LIN {X 0,Y 537.99,Z 256.093,A -85,B 0,C 180,E1 -3893.888,E2 -3893.888} C_VEL
LIN {X 0,Y 538.029,Z 256.085,A -85,B 0,C 180,E1 -3896.366,E2 -3896.366} C_VEL
LIN {X 0,Y 538.017,Z 256.09,A -85,B 0,C 180,E1 -3898.933,E2 -3898.933} C_VEL
LIN {X 0,Y 538.014,Z 256.089,A -85,B 0,C 180,E1 -3901.89,E2 -3901.89} C_VEL
LIN {X 0,Y 538.016,Z 256.087,A -85,B 0,C 180,E1 -3904.62,E2 -3904.62} C_VEL
LIN {X 0,Y 537.992,Z 256.097,A -85,B 0,C 180,E1 -3907.17,E2 -3907.17} C_VEL
LIN {X 0,Y 538.015,Z 256.09,A -85,B 0,C 180,E1 -3909.796,E2 -3909.796} C_VEL
LIN {X 0,Y 538.008,Z 256.09,A -85,B 0,C 180,E1 -3912.785,E2 -3912.785} C_VEL
LIN {X 0,Y 538.014,Z 256.088,A -85,B 0,C 180,E1 -3915.925,E2 -3915.925} C_VEL
LIN {X 0,Y 538.035,Z 256.094,A -85,B 0,C 180,E1 -3919.224,E2 -3919.224} C_VEL
LIN {X 0,Y 537.978,Z 256.092,A -85,B 0,C 180,E1 -3922.122,E2 -3922.122} C_VEL
LIN {X 0,Y 538,Z 256.094,A -85,B 0,C 180,E1 -3924.917,E2 -3924.917} C_VEL
LIN {X 0,Y 538.016,Z 256.09,A -85,B 0,C 180,E1 -3927.618,E2 -3927.618} C_VEL
LIN {X 0,Y 538.003,Z 256.088,A -85,B 0,C 180,E1 -3930.239,E2 -3930.239} C_VEL
LIN {X 0,Y 538.048,Z 256.087,A -85,B 0,C 180,E1 -3932.796,E2 -3932.796} C_VEL
LIN {X 0,Y 538.033,Z 256.092,A -85,B 0,C 180,E1 -3935.293,E2 -3935.293} C_VEL
LIN {X 0,Y 538.009,Z 256.089,A -85,B 0,C 180,E1 -3938.546,E2 -3938.546} C_VEL
LIN {X 0,Y 538.023,Z 256.092,A -85,B 0,C 180,E1 -3940.94,E2 -3940.94} C_VEL
LIN {X 0,Y 538.009,Z 256.094,A -85,B 0,C 180,E1 -3943.299,E2 -3943.299} C_VEL
LIN {X 0,Y 538.048,Z 256.085,A -85,B 0,C 180,E1 -3945.631,E2 -3945.631} C_VEL
LIN {X 0,Y 538.062,Z 256.085,A -85,B 0,C 180,E1 -3948.702,E2 -3948.702} C_VEL
LIN {X 0,Y 538.066,Z 256.082,A -85,B 0,C 180,E1 -3951.74,E2 -3951.74} C_VEL
LIN {X 0,Y 538.147,Z 256.075,A -85,B 0,C 180,E1 -3954.755,E2 -3954.755} C_VEL
LIN {X 0,Y 538.149,Z 256.071,A -85,B 0,C 180,E1 -3957.755,E2 -3957.755} C_VEL
LIN {X 0,Y 538.175,Z 256.072,A -85,B 0,C 180,E1 -3960.749,E2 -3960.749} C_VEL
LIN {X 0,Y 538.129,Z 256.083,A -85,B 0,C 180,E1 -3962.995,E2 -3962.995} C_VEL
LIN {X 0,Y 538.104,Z 256.076,A -85,B 0,C 180,E1 -3965.998,E2 -3965.998} C_VEL
LIN {X 0,Y 538.059,Z 256.09,A -85,B 0,C 180,E1 -3969.018,E2 -3969.018} C_VEL
LIN {X 0,Y 538.071,Z 256.08,A -85,B 0,C 180,E1 -3972.063,E2 -3972.063} C_VEL
LIN {X 0,Y 538.034,Z 256.091,A -85,B 0,C 180,E1 -3975.145,E2 -3975.145} C_VEL
LIN {X 0,Y 538.019,Z 256.088,A -85,B 0,C 180,E1 -3978.271,E2 -3978.271} C_VEL
LIN {X 0,Y 538.03,Z 256.091,A -85,B 0,C 180,E1 -3980.652,E2 -3980.652} C_VEL
LIN {X 0,Y 537.993,Z 256.09,A -85,B 0,C 180,E1 -3983.889,E2 -3983.889} C_VEL
LIN {X 0,Y 538.029,Z 256.088,A -85,B 0,C 180,E1 -3986.368,E2 -3986.368} C_VEL
LIN {X 0,Y 538.02,Z 256.095,A -85,B 0,C 180,E1 -3988.935,E2 -3988.935} C_VEL
LIN {X 0,Y 538,Z 256.089,A -85,B 0,C 180,E1 -3991.888,E2 -3991.888} C_VEL
LIN {X 0,Y 538.011,Z 256.094,A -85,B 0,C 180,E1 -3994.62,E2 -3994.62} C_VEL
LIN {X 0,Y 537.995,Z 256.093,A -85,B 0,C 180,E1 -3997.171,E2 -3997.171} C_VEL
LIN {X 0,Y 538.013,Z 256.087,A -85,B 0,C 180,E1 -3999.798,E2 -3999.798} C_VEL
LIN {X 0,Y 538.012,Z 256.097,A -85,B 0,C 180,E1 -4002.787,E2 -4002.787} C_VEL
LIN {X 0,Y 538.012,Z 256.088,A -85,B 0,C 180,E1 -4005.928,E2 -4005.928} C_VEL
LIN {X 0,Y 538.041,Z 256.087,A -85,B 0,C 180,E1 -4009.225,E2 -4009.225} C_VEL
LIN {X 0,Y 537.983,Z 256.093,A -85,B 0,C 180,E1 -4012.123,E2 -4012.123} C_VEL
LIN {X 0,Y 537.989,Z 256.096,A -85,B 0,C 180,E1 -4014.917,E2 -4014.917} C_VEL
LIN {X 0,Y 538.013,Z 256.088,A -85,B 0,C 180,E1 -4017.619,E2 -4017.619} C_VEL
LIN {X 0,Y 538.008,Z 256.095,A -85,B 0,C 180,E1 -4020.24,E2 -4020.24} C_VEL
LIN {X 0,Y 538.051,Z 256.188,A -85,B 0,C 180,E1 -4021.154,E2 -4021.154} C_VEL
LIN {X 0,Y 540.866,Z 268.014,A -85,B 0,C 180,E1 -4022.782,E2 -4022.782} C_VEL
LIN {X 0,Y 540.405,Z 289.739,A -85,B 0,C 180,E1 -4025.409,E2 -4025.409} C_VEL
LIN {X 0,Y 539.755,Z 315.114,A -85,B 0,C 180,E1 -4028.419,E2 -4028.419} C_VEL
LIN {X 0,Y 539.682,Z 320.744,A -85,B 0,C 180,E1 -4029.086,E2 -4029.086} C_VEL
LIN {X 0,Y 541.729,Z 333.165,A -85,B 0,C 180,E1 -4029.366,E2 -4029.366} C_VEL
LIN {X 0,Y 540.933,Z 482.028,A -85,B 0,C 180,E1 -4031.398,E2 -4031.398} C_VEL
LIN {X 0,Y 540.749,Z 497.284,A -85,B 0,C 180,E1 -4031.699,E2 -4031.699} C_VEL
LIN {X 0,Y 540.471,Z 512.684,A -85,B 0,C 180,E1 -4032.159,E2 -4032.159} C_VEL
LIN {X 0,Y 540.141,Z 526.944,A -85,B 0,C 180,E1 -4032.734,E2 -4032.734} C_VEL
LIN {X 0,Y 539.801,Z 540.926,A -85,B 0,C 180,E1 -4033.454,E2 -4033.454} C_VEL
LIN {X 0,Y 539.433,Z 554.517,A -85,B 0,C 180,E1 -4034.321,E2 -4034.321} C_VEL
LIN {X 0,Y 539.038,Z 566.884,A -85,B 0,C 180,E1 -4035.273,E2 -4035.273} C_VEL
LIN {X 0,Y 538.727,Z 577.285,A -85,B 0,C 180,E1 -4036.228,E2 -4036.228} C_VEL
LIN {X 0,Y 538.409,Z 587.775,A -85,B 0,C 180,E1 -4037.372,E2 -4037.372} C_VEL
LIN {X 0,Y 538.086,Z 598.023,A -85,B 0,C 180,E1 -4038.703,E2 -4038.703} C_VEL
LIN {X 0,Y 537.901,Z 606.538,A -85,B 0,C 180,E1 -4040.032,E2 -4040.032} C_VEL
LIN {X 0,Y 537.748,Z 613.621,A -85,B 0,C 180,E1 -4041.357,E2 -4041.357} C_VEL
LIN {X 0,Y 537.647,Z 620.187,A -85,B 0,C 180,E1 -4042.868,E2 -4042.868} C_VEL
LIN {X 0,Y 537.641,Z 625.323,A -85,B 0,C 180,E1 -4044.375,E2 -4044.375} C_VEL
LIN {X 0,Y 537.507,Z 628.293,A -85,B 0,C 180,E1 -4045.502,E2 -4045.502} C_VEL
LIN {X 0,Y 537.544,Z 631.186,A -85,B 0,C 180,E1 -4047.003,E2 -4047.003} C_VEL
LIN {X 0,Y 537.449,Z 632.91,A -85,B 0,C 180,E1 -4048.502,E2 -4048.502} C_VEL
LIN {X 0,Y 537.439,Z 633.5,A -85,B 0,C 180,E1 -4050.001,E2 -4050.001} C_VEL
LIN {X 0,Y 537.449,Z 632.906,A -85,B 0,C 180,E1 -4051.5,E2 -4051.5} C_VEL
LIN {X 0,Y 537.544,Z 631.178,A -85,B 0,C 180,E1 -4052.999,E2 -4052.999} C_VEL
LIN {X 0,Y 537.507,Z 628.286,A -85,B 0,C 180,E1 -4054.501,E2 -4054.501} C_VEL
LIN {X 0,Y 537.619,Z 624.162,A -85,B 0,C 180,E1 -4056.004,E2 -4056.004} C_VEL
LIN {X 0,Y 537.663,Z 618.696,A -85,B 0,C 180,E1 -4057.512,E2 -4057.512} C_VEL
LIN {X 0,Y 537.798,Z 611.738,A -85,B 0,C 180,E1 -4059.023,E2 -4059.023} C_VEL
LIN {X 0,Y 538.025,Z 603.074,A -85,B 0,C 180,E1 -4060.538,E2 -4060.538} C_VEL
LIN {X 0,Y 538.231,Z 593.526,A -85,B 0,C 180,E1 -4061.913,E2 -4061.913} C_VEL
LIN {X 0,Y 538.526,Z 584.5,A -85,B 0,C 180,E1 -4063.011,E2 -4063.011} C_VEL
LIN {X 0,Y 538.805,Z 573.332,A -85,B 0,C 180,E1 -4064.157,E2 -4064.157} C_VEL
LIN {X 0,Y 539.214,Z 561.283,A -85,B 0,C 180,E1 -4065.175,E2 -4065.175} C_VEL
LIN {X 0,Y 539.564,Z 548.573,A -85,B 0,C 180,E1 -4066.069,E2 -4066.069} C_VEL
LIN {X 0,Y 539.958,Z 535.353,A -85,B 0,C 180,E1 -4066.835,E2 -4066.835} C_VEL
LIN {X 0,Y 540.222,Z 522.073,A -85,B 0,C 180,E1 -4067.46,E2 -4067.46} C_VEL
LIN {X 0,Y 540.55,Z 506.912,A -85,B 0,C 180,E1 -4068.012,E2 -4068.012} C_VEL
LIN {X 0,Y 540.767,Z 490.824,A -85,B 0,C 180,E1 -4068.426,E2 -4068.426} C_VEL
LIN {X 0,Y 540.951,Z 468.028,A -85,B 0,C 180,E1 -4068.778,E2 -4068.778} C_VEL
LIN {X 0,Y 541.696,Z 333.032,A -85,B 0,C 180,E1 -4070.627,E2 -4070.627} C_VEL
LIN {X 0,Y 539.547,Z 319.836,A -85,B 0,C 180,E1 -4070.932,E2 -4070.932} C_VEL
LIN {X 0,Y 539.988,Z 295.22,A -85,B 0,C 180,E1 -4073.796,E2 -4073.796} C_VEL
LIN {X 0,Y 540.451,Z 272.845,A -85,B 0,C 180,E1 -4076.449,E2 -4076.449} C_VEL
LIN {X 0,Y 540.417,Z 266.435,A -85,B 0,C 180,E1 -4077.227,E2 -4077.227} C_VEL
LIN {X 0,Y 538.042,Z 256.092,A -85,B 0,C 180,E1 -4078.635,E2 -4078.635} C_VEL
LIN {X 0,Y 538.013,Z 256.096,A -85,B 0,C 180,E1 -4081.502,E2 -4081.502} C_VEL
LIN {X 0,Y 538.022,Z 256.09,A -85,B 0,C 180,E1 -4084.174,E2 -4084.174} C_VEL
LIN {X 0,Y 538.009,Z 256.097,A -85,B 0,C 180,E1 -4087.17,E2 -4087.17} C_VEL
LIN {X 0,Y 538.03,Z 256.088,A -85,B 0,C 180,E1 -4089.797,E2 -4089.797} C_VEL
LIN {X 0,Y 538.024,Z 256.095,A -85,B 0,C 180,E1 -4092.786,E2 -4092.786} C_VEL
LIN {X 0,Y 538.029,Z 256.088,A -85,B 0,C 180,E1 -4095.926,E2 -4095.926} C_VEL
LIN {X 0,Y 538.054,Z 256.086,A -85,B 0,C 180,E1 -4099.224,E2 -4099.224} C_VEL
LIN {X 0,Y 537.994,Z 256.094,A -85,B 0,C 180,E1 -4102.122,E2 -4102.122} C_VEL
LIN {X 0,Y 538,Z 256.095,A -85,B 0,C 180,E1 -4104.915,E2 -4104.915} C_VEL
LIN {X 0,Y 538.025,Z 256.089,A -85,B 0,C 180,E1 -4107.617,E2 -4107.617} C_VEL
LIN {X 0,Y 538.019,Z 256.096,A -85,B 0,C 180,E1 -4110.239,E2 -4110.239} C_VEL
LIN {X 0,Y 538.038,Z 256.091,A -85,B 0,C 180,E1 -4112.794,E2 -4112.794} C_VEL
LIN {X 0,Y 538.028,Z 256.091,A -85,B 0,C 180,E1 -4115.291,E2 -4115.291} C_VEL
LIN {X 0,Y 538.035,Z 256.167,A -85,B 0,C 180,E1 -4117.512,E2 -4117.512} C_VEL
LIN {X 0,Y 539.535,Z 263.399,A -85,B 0,C 180,E1 -4118.809,E2 -4118.809} C_VEL
LIN {X 0,Y 539.458,Z 265.534,A -85,B 0,C 180,E1 -4119.16,E2 -4119.16} C_VEL
LIN {X 0,Y 541.828,Z 276.302,A -85,B 0,C 180,E1 -4119.422,E2 -4119.422} C_VEL
LIN {X 0,Y 540.818,Z 430.376,A -85,B 0,C 180,E1 -4121.6,E2 -4121.6} C_VEL
LIN {X 0,Y 540.6,Z 446.158,A -85,B 0,C 180,E1 -4121.991,E2 -4121.991} C_VEL
LIN {X 0,Y 540.318,Z 460.654,A -85,B 0,C 180,E1 -4122.494,E2 -4122.494} C_VEL
LIN {X 0,Y 539.979,Z 475.113,A -85,B 0,C 180,E1 -4123.166,E2 -4123.166} C_VEL
LIN {X 0,Y 539.634,Z 488.397,A -85,B 0,C 180,E1 -4123.933,E2 -4123.933} C_VEL
LIN {X 0,Y 539.235,Z 501.769,A -85,B 0,C 180,E1 -4124.89,E2 -4124.89} C_VEL
LIN {X 0,Y 538.856,Z 512.924,A -85,B 0,C 180,E1 -4125.845,E2 -4125.845} C_VEL
LIN {X 0,Y 538.54,Z 524.137,A -85,B 0,C 180,E1 -4126.99,E2 -4126.99} C_VEL
LIN {X 0,Y 538.257,Z 533.189,A -85,B 0,C 180,E1 -4128.088,E2 -4128.088} C_VEL
LIN {X 0,Y 538.063,Z 541.564,A -85,B 0,C 180,E1 -4129.273,E2 -4129.273} C_VEL
LIN {X 0,Y 537.827,Z 549.47,A -85,B 0,C 180,E1 -4130.599,E2 -4130.599} C_VEL
LIN {X 0,Y 537.732,Z 555.16,A -85,B 0,C 180,E1 -4131.734,E2 -4131.734} C_VEL
LIN {X 0,Y 537.653,Z 559.975,A -85,B 0,C 180,E1 -4132.866,E2 -4132.866} C_VEL
LIN {X 0,Y 537.643,Z 565.194,A -85,B 0,C 180,E1 -4134.373,E2 -4134.373} C_VEL
LIN {X 0,Y 537.507,Z 568.211,A -85,B 0,C 180,E1 -4135.5,E2 -4135.5} C_VEL
LIN {X 0,Y 537.545,Z 571.096,A -85,B 0,C 180,E1 -4137.002,E2 -4137.002} C_VEL
LIN {X 0,Y 537.45,Z 572.839,A -85,B 0,C 180,E1 -4138.501,E2 -4138.501} C_VEL
LIN {X 0,Y 537.438,Z 573.496,A -85,B 0,C 180,E1 -4139.999,E2 -4139.999} C_VEL
LIN {X 0,Y 537.449,Z 572.919,A -85,B 0,C 180,E1 -4141.498,E2 -4141.498} C_VEL
LIN {X 0,Y 537.546,Z 571.231,A -85,B 0,C 180,E1 -4142.997,E2 -4142.997} C_VEL
LIN {X 0,Y 537.508,Z 568.43,A -85,B 0,C 180,E1 -4144.499,E2 -4144.499} C_VEL
LIN {X 0,Y 537.596,Z 564.272,A -85,B 0,C 180,E1 -4146.003,E2 -4146.003} C_VEL
LIN {X 0,Y 537.649,Z 560.325,A -85,B 0,C 180,E1 -4147.133,E2 -4147.133} C_VEL
LIN {X 0,Y 537.745,Z 553.861,A -85,B 0,C 180,E1 -4148.644,E2 -4148.644} C_VEL
LIN {X 0,Y 537.9,Z 546.786,A -85,B 0,C 180,E1 -4149.969,E2 -4149.969} C_VEL
LIN {X 0,Y 538.081,Z 539.601,A -85,B 0,C 180,E1 -4151.107,E2 -4151.107} C_VEL
LIN {X 0,Y 538.284,Z 531.285,A -85,B 0,C 180,E1 -4152.249,E2 -4152.249} C_VEL
LIN {X 0,Y 538.608,Z 521.487,A -85,B 0,C 180,E1 -4153.391,E2 -4153.391} C_VEL
LIN {X 0,Y 538.964,Z 509.674,A -85,B 0,C 180,E1 -4154.537,E2 -4154.537} C_VEL
LIN {X 0,Y 539.401,Z 496.451,A -85,B 0,C 180,E1 -4155.606,E2 -4155.606} C_VEL
LIN {X 0,Y 539.759,Z 483.659,A -85,B 0,C 180,E1 -4156.45,E2 -4156.45} C_VEL
LIN {X 0,Y 540.171,Z 469.437,A -85,B 0,C 180,E1 -4157.216,E2 -4157.216} C_VEL
LIN {X 0,Y 540.457,Z 455.669,A -85,B 0,C 180,E1 -4157.793,E2 -4157.793} C_VEL
LIN {X 0,Y 540.708,Z 440.867,A -85,B 0,C 180,E1 -4158.267,E2 -4158.267} C_VEL
LIN {X 0,Y 540.889,Z 426.516,A -85,B 0,C 180,E1 -4158.575,E2 -4158.575} C_VEL
LIN {X 0,Y 541.778,Z 281.95,A -85,B 0,C 180,E1 -4160.585,E2 -4160.585} C_VEL
LIN {X 0,Y 541.216,Z 277.894,A -85,B 0,C 180,E1 -4160.68,E2 -4160.68} C_VEL
LIN {X 0,Y 539.647,Z 274.151,A -85,B 0,C 180,E1 -4160.807,E2 -4160.807} C_VEL
LIN {X 0,Y 534.961,Z 267.695,A -85,B 0,C 180,E1 -4161.077,E2 -4161.077} C_VEL
LIN {X 0,Y 532.571,Z 264.733,A -85,B 0,C 180,E1 -4161.255,E2 -4161.255} C_VEL
LIN {X 0,Y 532.357,Z 264.168,A -85,B 0,C 180,E1 -4161.327,E2 -4161.327} C_VEL
LIN {X 0,Y 530.972,Z 256.972,A -85,B 0,C 180,E1 -4162.597,E2 -4162.597} C_VEL
LIN {X 0,Y 530.971,Z 256.973,A -85,B 0,C 180,E1 -4165.833,E2 -4165.833} C_VEL
LIN {X 0,Y 530.968,Z 256.968,A -85,B 0,C 180,E1 -4168.456,E2 -4168.456} C_VEL
LIN {X 0,Y 530.953,Z 256.968,A -85,B 0,C 180,E1 -4171.078,E2 -4171.078} C_VEL
LIN {X 0,Y 530.986,Z 256.97,A -85,B 0,C 180,E1 -4173.772,E2 -4173.772} C_VEL
LIN {X 0,Y 530.949,Z 256.968,A -85,B 0,C 180,E1 -4176.558,E2 -4176.558} C_VEL
LIN {X 0,Y 530.984,Z 256.966,A -85,B 0,C 180,E1 -4179.442,E2 -4179.442} C_VEL
LIN {X 0,Y 530.972,Z 256.966,A -85,B 0,C 180,E1 -4182.456,E2 -4182.456} C_VEL
LIN {X 0,Y 530.974,Z 256.97,A -85,B 0,C 180,E1 -4185.621,E2 -4185.621} C_VEL
LIN {X 0,Y 530.991,Z 256.962,A -85,B 0,C 180,E1 -4188.563,E2 -4188.563} C_VEL
LIN {X 0,Y 530.953,Z 256.972,A -85,B 0,C 180,E1 -4191.528,E2 -4191.528} C_VEL
LIN {X 0,Y 530.951,Z 256.968,A -85,B 0,C 180,E1 -4194.379,E2 -4194.379} C_VEL
LIN {X 0,Y 530.962,Z 256.967,A -85,B 0,C 180,E1 -4197.132,E2 -4197.132} C_VEL
LIN {X 0,Y 530.965,Z 256.974,A -85,B 0,C 180,E1 -4199.802,E2 -4199.802} C_VEL
LIN {X 0,Y 530.97,Z 256.965,A -85,B 0,C 180,E1 -4202.474,E2 -4202.474} C_VEL
LIN {X 0,Y 530.983,Z 256.963,A -85,B 0,C 180,E1 -4204.94,E2 -4204.94} C_VEL
LIN {X 0,Y 530.965,Z 256.967,A -85,B 0,C 180,E1 -4208.246,E2 -4208.246} C_VEL
LIN {X 0,Y 530.986,Z 256.962,A -85,B 0,C 180,E1 -4210.676,E2 -4210.676} C_VEL
LIN {X 0,Y 530.97,Z 256.966,A -85,B 0,C 180,E1 -4213.07,E2 -4213.07} C_VEL
LIN {X 0,Y 531.012,Z 256.966,A -85,B 0,C 180,E1 -4215.435,E2 -4215.435} C_VEL
LIN {X 0,Y 531.03,Z 256.957,A -85,B 0,C 180,E1 -4218.549,E2 -4218.549} C_VEL
LIN {X 0,Y 531.048,Z 256.964,A -85,B 0,C 180,E1 -4221.628,E2 -4221.628} C_VEL
LIN {X 0,Y 531.111,Z 256.947,A -85,B 0,C 180,E1 -4224.684,E2 -4224.684} C_VEL
LIN {X 0,Y 531.127,Z 256.952,A -85,B 0,C 180,E1 -4227.724,E2 -4227.724} C_VEL
LIN {X 0,Y 531.144,Z 256.943,A -85,B 0,C 180,E1 -4230.757,E2 -4230.757} C_VEL
LIN {X 0,Y 531.096,Z 256.951,A -85,B 0,C 180,E1 -4233.033,E2 -4233.033} C_VEL
LIN {X 0,Y 531.065,Z 256.955,A -85,B 0,C 180,E1 -4236.076,E2 -4236.076} C_VEL
LIN {X 0,Y 531.04,Z 256.956,A -85,B 0,C 180,E1 -4238.37,E2 -4238.37} C_VEL
LIN {X 0,Y 531.04,Z 256.962,A -85,B 0,C 180,E1 -4241.671,E2 -4241.671} C_VEL
LIN {X 0,Y 531.019,Z 256.961,A -85,B 0,C 180,E1 -4244.955,E2 -4244.955} C_VEL
LIN {X 0,Y 531.005,Z 256.965,A -85,B 0,C 180,E1 -4247.721,E2 -4247.721} C_VEL
LIN {X 0,Y 530.987,Z 256.965,A -85,B 0,C 180,E1 -4250.937,E2 -4250.937} C_VEL
LIN {X 0,Y 530.952,Z 256.967,A -85,B 0,C 180,E1 -4254.224,E2 -4254.224} C_VEL
LIN {X 0,Y 530.991,Z 256.963,A -85,B 0,C 180,E1 -4256.743,E2 -4256.743} C_VEL
LIN {X 0,Y 530.968,Z 256.974,A -85,B 0,C 180,E1 -4259.322,E2 -4259.322} C_VEL
LIN {X 0,Y 530.966,Z 256.966,A -85,B 0,C 180,E1 -4262.102,E2 -4262.102} C_VEL
LIN {X 0,Y 530.973,Z 256.967,A -85,B 0,C 180,E1 -4264.853,E2 -4264.853} C_VEL
LIN {X 0,Y 530.952,Z 256.974,A -85,B 0,C 180,E1 -4267.507,E2 -4267.507} C_VEL
LIN {X 0,Y 530.97,Z 256.965,A -85,B 0,C 180,E1 -4270.432,E2 -4270.432} C_VEL
LIN {X 0,Y 530.951,Z 256.973,A -85,B 0,C 180,E1 -4273.494,E2 -4273.494} C_VEL
LIN {X 0,Y 530.951,Z 256.967,A -85,B 0,C 180,E1 -4276.505,E2 -4276.505} C_VEL
LIN {X 0,Y 530.969,Z 256.969,A -85,B 0,C 180,E1 -4279.567,E2 -4279.567} C_VEL
LIN {X 0,Y 530.953,Z 256.968,A -85,B 0,C 180,E1 -4282.577,E2 -4282.577} C_VEL
LIN {X 0,Y 530.984,Z 256.971,A -85,B 0,C 180,E1 -4285.311,E2 -4285.311} C_VEL
LIN {X 0,Y 530.967,Z 256.965,A -85,B 0,C 180,E1 -4288.033,E2 -4288.033} C_VEL
LIN {X 0,Y 530.973,Z 256.969,A -85,B 0,C 180,E1 -4290.874,E2 -4290.874} C_VEL
LIN {X 0,Y 530.989,Z 256.971,A -85,B 0,C 180,E1 -4293.256,E2 -4293.256} C_VEL
LIN {X 0,Y 530.97,Z 256.965,A -85,B 0,C 180,E1 -4295.961,E2 -4295.961} C_VEL
LIN {X 0,Y 530.987,Z 256.971,A -85,B 0,C 180,E1 -4299.062,E2 -4299.062} C_VEL
LIN {X 0,Y 531.002,Z 256.961,A -85,B 0,C 180,E1 -4302.278,E2 -4302.278} C_VEL
LIN {X 0,Y 531.004,Z 256.965,A -85,B 0,C 180,E1 -4305.436,E2 -4305.436} C_VEL
LIN {X 0,Y 531.022,Z 256.96,A -85,B 0,C 180,E1 -4308.55,E2 -4308.55} C_VEL
LIN {X 0,Y 531.036,Z 256.958,A -85,B 0,C 180,E1 -4311.63,E2 -4311.63} C_VEL
LIN {X 0,Y 531.106,Z 256.952,A -85,B 0,C 180,E1 -4314.686,E2 -4314.686} C_VEL
LIN {X 0,Y 531.121,Z 256.947,A -85,B 0,C 180,E1 -4317.726,E2 -4317.726} C_VEL
LIN {X 0,Y 531.144,Z 256.948,A -85,B 0,C 180,E1 -4320.759,E2 -4320.759} C_VEL
LIN {X 0,Y 531.094,Z 256.958,A -85,B 0,C 180,E1 -4323.035,E2 -4323.035} C_VEL
LIN {X 0,Y 531.06,Z 256.953,A -85,B 0,C 180,E1 -4326.078,E2 -4326.078} C_VEL
LIN {X 0,Y 531.044,Z 256.957,A -85,B 0,C 180,E1 -4328.371,E2 -4328.371} C_VEL
LIN {X 0,Y 531.042,Z 256.956,A -85,B 0,C 180,E1 -4331.674,E2 -4331.674} C_VEL
LIN {X 0,Y 531.019,Z 256.968,A -85,B 0,C 180,E1 -4334.957,E2 -4334.957} C_VEL
LIN {X 0,Y 531.005,Z 256.961,A -85,B 0,C 180,E1 -4337.723,E2 -4337.723} C_VEL
LIN {X 0,Y 530.99,Z 256.971,A -85,B 0,C 180,E1 -4340.939,E2 -4340.939} C_VEL
LIN {X 0,Y 530.959,Z 256.967,A -85,B 0,C 180,E1 -4344.226,E2 -4344.226} C_VEL
LIN {X 0,Y 530.989,Z 256.97,A -85,B 0,C 180,E1 -4346.745,E2 -4346.745} C_VEL
LIN {X 0,Y 530.971,Z 256.967,A -85,B 0,C 180,E1 -4349.324,E2 -4349.324} C_VEL
LIN {X 0,Y 530.955,Z 256.967,A -85,B 0,C 180,E1 -4352.101,E2 -4352.101} C_VEL
LIN {X 0,Y 530.967,Z 256.974,A -85,B 0,C 180,E1 -4354.853,E2 -4354.853} C_VEL
LIN {X 0,Y 530.956,Z 256.967,A -85,B 0,C 180,E1 -4357.509,E2 -4357.509} C_VEL
LIN {X 0,Y 530.972,Z 256.969,A -85,B 0,C 180,E1 -4360.434,E2 -4360.434} C_VEL
LIN {X 0,Y 530.952,Z 256.969,A -85,B 0,C 180,E1 -4363.282,E2 -4363.282} C_VEL
LIN {X 0,Y 530.97,Z 256.965,A -85,B 0,C 180,E1 -4365.623,E2 -4365.623} C_VEL
LIN {X 0,Y 530.986,Z 256.97,A -85,B 0,C 180,E1 -4368.566,E2 -4368.566} C_VEL
LIN {X 0,Y 530.95,Z 256.968,A -85,B 0,C 180,E1 -4371.531,E2 -4371.531} C_VEL
LIN {X 0,Y 530.944,Z 256.973,A -85,B 0,C 180,E1 -4374.381,E2 -4374.381} C_VEL
LIN {X 0,Y 530.962,Z 256.97,A -85,B 0,C 180,E1 -4377.135,E2 -4377.135} C_VEL
LIN {X 0,Y 530.956,Z 256.971,A -85,B 0,C 180,E1 -4379.804,E2 -4379.804} C_VEL
LIN {X 0,Y 530.983,Z 257.021,A -85,B 0,C 180,E1 -4380.876,E2 -4380.876} C_VEL
LIN {X 0,Y 533.946,Z 269.092,A -85,B 0,C 180,E1 -4382.57,E2 -4382.57} C_VEL
LIN {X 0,Y 533.882,Z 277.85,A -85,B 0,C 180,E1 -4383.657,E2 -4383.657} C_VEL
LIN {X 0,Y 533.271,Z 301.309,A -85,B 0,C 180,E1 -4386.507,E2 -4386.507} C_VEL
LIN {X 0,Y 532.798,Z 320.695,A -85,B 0,C 180,E1 -4388.816,E2 -4388.816} C_VEL
LIN {X 0,Y 535.075,Z 334.407,A -85,B 0,C 180,E1 -4389.122,E2 -4389.122} C_VEL
LIN {X 0,Y 534.178,Z 478.803,A -85,B 0,C 180,E1 -4391.133,E2 -4391.133} C_VEL
LIN {X 0,Y 533.983,Z 495.281,A -85,B 0,C 180,E1 -4391.44,E2 -4391.44} C_VEL
LIN {X 0,Y 533.681,Z 510.286,A -85,B 0,C 180,E1 -4391.875,E2 -4391.875} C_VEL
LIN {X 0,Y 533.284,Z 524.99,A -85,B 0,C 180,E1 -4392.456,E2 -4392.456} C_VEL
LIN {X 0,Y 532.92,Z 540.126,A -85,B 0,C 180,E1 -4393.234,E2 -4393.234} C_VEL
LIN {X 0,Y 532.481,Z 553.999,A -85,B 0,C 180,E1 -4394.126,E2 -4394.126} C_VEL
LIN {X 0,Y 532.037,Z 567.313,A -85,B 0,C 180,E1 -4395.172,E2 -4395.172} C_VEL
LIN {X 0,Y 531.652,Z 578.65,A -85,B 0,C 180,E1 -4396.236,E2 -4396.236} C_VEL
LIN {X 0,Y 531.346,Z 589.057,A -85,B 0,C 180,E1 -4397.395,E2 -4397.395} C_VEL
LIN {X 0,Y 531.055,Z 599.228,A -85,B 0,C 180,E1 -4398.745,E2 -4398.745} C_VEL
LIN {X 0,Y 530.808,Z 607.644,A -85,B 0,C 180,E1 -4400.09,E2 -4400.09} C_VEL
LIN {X 0,Y 530.664,Z 615.428,A -85,B 0,C 180,E1 -4401.624,E2 -4401.624} C_VEL
LIN {X 0,Y 530.549,Z 621.61,A -85,B 0,C 180,E1 -4403.154,E2 -4403.154} C_VEL
LIN {X 0,Y 530.508,Z 626.388,A -85,B 0,C 180,E1 -4404.68,E2 -4404.68} C_VEL
LIN {X 0,Y 530.48,Z 629.888,A -85,B 0,C 180,E1 -4406.203,E2 -4406.203} C_VEL
LIN {X 0,Y 530.408,Z 632.19,A -85,B 0,C 180,E1 -4407.723,E2 -4407.723} C_VEL
LIN {X 0,Y 530.342,Z 633.348,A -85,B 0,C 180,E1 -4409.242,E2 -4409.242} C_VEL
LIN {X 0,Y 530.342,Z 633.346,A -85,B 0,C 180,E1 -4410.76,E2 -4410.76} C_VEL
LIN {X 0,Y 530.408,Z 632.184,A -85,B 0,C 180,E1 -4412.279,E2 -4412.279} C_VEL
LIN {X 0,Y 530.48,Z 629.88,A -85,B 0,C 180,E1 -4413.799,E2 -4413.799} C_VEL
LIN {X 0,Y 530.509,Z 626.384,A -85,B 0,C 180,E1 -4415.322,E2 -4415.322} C_VEL
LIN {X 0,Y 530.551,Z 621.605,A -85,B 0,C 180,E1 -4416.848,E2 -4416.848} C_VEL
LIN {X 0,Y 530.666,Z 615.415,A -85,B 0,C 180,E1 -4418.378,E2 -4418.378} C_VEL
LIN {X 0,Y 530.809,Z 607.625,A -85,B 0,C 180,E1 -4419.912,E2 -4419.912} C_VEL
LIN {X 0,Y 531.052,Z 600.483,A -85,B 0,C 180,E1 -4421.064,E2 -4421.064} C_VEL
LIN {X 0,Y 531.295,Z 590.527,A -85,B 0,C 180,E1 -4422.414,E2 -4422.414} C_VEL
LIN {X 0,Y 531.6,Z 580.316,A -85,B 0,C 180,E1 -4423.573,E2 -4423.573} C_VEL
LIN {X 0,Y 531.974,Z 568.153,A -85,B 0,C 180,E1 -4424.734,E2 -4424.734} C_VEL
LIN {X 0,Y 532.372,Z 555.984,A -85,B 0,C 180,E1 -4425.702,E2 -4425.702} C_VEL
LIN {X 0,Y 532.762,Z 542.763,A -85,B 0,C 180,E1 -4426.576,E2 -4426.576} C_VEL
LIN {X 0,Y 533.119,Z 528.248,A -85,B 0,C 180,E1 -4427.354,E2 -4427.354} C_VEL
LIN {X 0,Y 533.537,Z 513.145,A -85,B 0,C 180,E1 -4427.984,E2 -4427.984} C_VEL
LIN {X 0,Y 533.839,Z 497.967,A -85,B 0,C 180,E1 -4428.452,E2 -4428.452} C_VEL
LIN {X 0,Y 534.047,Z 483.066,A -85,B 0,C 180,E1 -4428.763,E2 -4428.763} C_VEL
LIN {X 0,Y 535.025,Z 333.867,A -85,B 0,C 180,E1 -4430.873,E2 -4430.873} C_VEL
LIN {X 0,Y 532.621,Z 319.288,A -85,B 0,C 180,E1 -4431.208,E2 -4431.208} C_VEL
LIN {X 0,Y 533.097,Z 296.352,A -85,B 0,C 180,E1 -4433.916,E2 -4433.916} C_VEL
LIN {X 0,Y 533.634,Z 274.064,A -85,B 0,C 180,E1 -4436.602,E2 -4436.602} C_VEL
LIN {X 0,Y 533.705,Z 268.95,A -85,B 0,C 180,E1 -4437.233,E2 -4437.233} C_VEL
LIN {X 0,Y 530.989,Z 256.971,A -85,B 0,C 180,E1 -4438.914,E2 -4438.914} C_VEL
LIN {X 0,Y 530.97,Z 256.97,A -85,B 0,C 180,E1 -4442.101,E2 -4442.101} C_VEL
LIN {X 0,Y 530.974,Z 256.973,A -85,B 0,C 180,E1 -4444.851,E2 -4444.851} C_VEL
LIN {X 0,Y 530.971,Z 256.97,A -85,B 0,C 180,E1 -4447.508,E2 -4447.508} C_VEL
LIN {X 0,Y 530.987,Z 256.968,A -85,B 0,C 180,E1 -4450.433,E2 -4450.433} C_VEL
LIN {X 0,Y 530.966,Z 256.971,A -85,B 0,C 180,E1 -4453.281,E2 -4453.281} C_VEL
LIN {X 0,Y 530.99,Z 256.965,A -85,B 0,C 180,E1 -4455.621,E2 -4455.621} C_VEL
LIN {X 0,Y 530.999,Z 256.97,A -85,B 0,C 180,E1 -4458.565,E2 -4458.565} C_VEL
LIN {X 0,Y 530.959,Z 256.968,A -85,B 0,C 180,E1 -4461.529,E2 -4461.529} C_VEL
LIN {X 0,Y 530.956,Z 256.975,A -85,B 0,C 180,E1 -4464.38,E2 -4464.38} C_VEL
LIN {X 0,Y 530.973,Z 256.968,A -85,B 0,C 180,E1 -4467.133,E2 -4467.133} C_VEL
LIN {X 0,Y 530.974,Z 256.969,A -85,B 0,C 180,E1 -4469.803,E2 -4469.803} C_VEL
LIN {X 0,Y 530.979,Z 256.972,A -85,B 0,C 180,E1 -4472.476,E2 -4472.476} C_VEL
LIN {X 0,Y 530.994,Z 256.968,A -85,B 0,C 180,E1 -4474.941,E2 -4474.941} C_VEL
LIN {X 0,Y 530.984,Z 257.09,A -85,B 0,C 180,E1 -4477.248,E2 -4477.248} C_VEL
LIN {X 0,Y 532.712,Z 265.192,A -85,B 0,C 180,E1 -4478.727,E2 -4478.727} C_VEL
LIN {X 0,Y 532.725,Z 266.422,A -85,B 0,C 180,E1 -4478.899,E2 -4478.899} C_VEL
LIN {X 0,Y 535.172,Z 276.789,A -85,B 0,C 180,E1 -4479.161,E2 -4479.161} C_VEL
LIN {X 0,Y 534.114,Z 420.858,A -85,B 0,C 180,E1 -4481.232,E2 -4481.232} C_VEL
LIN {X 0,Y 533.962,Z 436.84,A -85,B 0,C 180,E1 -4481.527,E2 -4481.527} C_VEL
LIN {X 0,Y 533.704,Z 452.36,A -85,B 0,C 180,E1 -4481.973,E2 -4481.973} C_VEL
LIN {X 0,Y 533.343,Z 466.942,A -85,B 0,C 180,E1 -4482.555,E2 -4482.555} C_VEL
LIN {X 0,Y 532.949,Z 481.975,A -85,B 0,C 180,E1 -4483.332,E2 -4483.332} C_VEL
LIN {X 0,Y 532.517,Z 495.793,A -85,B 0,C 180,E1 -4484.233,E2 -4484.233} C_VEL
LIN {X 0,Y 532.073,Z 508.788,A -85,B 0,C 180,E1 -4485.269,E2 -4485.269} C_VEL
LIN {X 0,Y 531.755,Z 518.919,A -85,B 0,C 180,E1 -4486.237,E2 -4486.237} C_VEL
LIN {X 0,Y 531.385,Z 529.267,A -85,B 0,C 180,E1 -4487.395,E2 -4487.395} C_VEL
LIN {X 0,Y 531.086,Z 539.272,A -85,B 0,C 180,E1 -4488.744,E2 -4488.744} C_VEL
LIN {X 0,Y 530.906,Z 546.479,A -85,B 0,C 180,E1 -4489.898,E2 -4489.898} C_VEL
LIN {X 0,Y 530.693,Z 553.611,A -85,B 0,C 180,E1 -4491.24,E2 -4491.24} C_VEL
LIN {X 0,Y 530.575,Z 560.09,A -85,B 0,C 180,E1 -4492.77,E2 -4492.77} C_VEL
LIN {X 0,Y 530.551,Z 565.23,A -85,B 0,C 180,E1 -4494.298,E2 -4494.298} C_VEL
LIN {X 0,Y 530.412,Z 568.208,A -85,B 0,C 180,E1 -4495.44,E2 -4495.44} C_VEL
LIN {X 0,Y 530.45,Z 571.093,A -85,B 0,C 180,E1 -4496.962,E2 -4496.962} C_VEL
LIN {X 0,Y 530.407,Z 572.162,A -85,B 0,C 180,E1 -4497.721,E2 -4497.721} C_VEL
LIN {X 0,Y 530.341,Z 573.286,A -85,B 0,C 180,E1 -4499.24,E2 -4499.24} C_VEL
LIN {X 0,Y 530.339,Z 573.496,A -85,B 0,C 180,E1 -4499.999,E2 -4499.999} C_VEL
LIN {X 0,Y 530.359,Z 572.913,A -85,B 0,C 180,E1 -4501.518,E2 -4501.518} C_VEL
LIN {X 0,Y 530.409,Z 572.269,A -85,B 0,C 180,E1 -4502.278,E2 -4502.278} C_VEL
LIN {X 0,Y 530.483,Z 569.954,A -85,B 0,C 180,E1 -4503.798,E2 -4503.798} C_VEL
LIN {X 0,Y 530.413,Z 568.431,A -85,B 0,C 180,E1 -4504.559,E2 -4504.559} C_VEL
LIN {X 0,Y 530.506,Z 564.311,A -85,B 0,C 180,E1 -4506.083,E2 -4506.083} C_VEL
LIN {X 0,Y 530.599,Z 558.971,A -85,B 0,C 180,E1 -4507.611,E2 -4507.611} C_VEL
LIN {X 0,Y 530.748,Z 552.101,A -85,B 0,C 180,E1 -4509.142,E2 -4509.142} C_VEL
LIN {X 0,Y 530.969,Z 544.711,A -85,B 0,C 180,E1 -4510.485,E2 -4510.485} C_VEL
LIN {X 0,Y 531.201,Z 535.513,A -85,B 0,C 180,E1 -4511.878,E2 -4511.878} C_VEL
LIN {X 0,Y 531.479,Z 526.695,A -85,B 0,C 180,E1 -4512.99,E2 -4512.99} C_VEL
LIN {X 0,Y 531.849,Z 515.962,A -85,B 0,C 180,E1 -4514.149,E2 -4514.149} C_VEL
LIN {X 0,Y 532.27,Z 504.1,A -85,B 0,C 180,E1 -4515.213,E2 -4515.213} C_VEL
LIN {X 0,Y 532.66,Z 491.179,A -85,B 0,C 180,E1 -4516.183,E2 -4516.183} C_VEL
LIN {X 0,Y 533.157,Z 476.767,A -85,B 0,C 180,E1 -4517.055,E2 -4517.055} C_VEL
LIN {X 0,Y 533.471,Z 462.701,A -85,B 0,C 180,E1 -4517.736,E2 -4517.736} C_VEL
LIN {X 0,Y 533.768,Z 447.471,A -85,B 0,C 180,E1 -4518.296,E2 -4518.296} C_VEL
LIN {X 0,Y 534.072,Z 432.322,A -85,B 0,C 180,E1 -4518.691,E2 -4518.691} C_VEL
LIN {X 0,Y 534.262,Z 406.024,A -85,B 0,C 180,E1 -4519.103,E2 -4519.103} C_VEL
LIN {X 0,Y 535.182,Z 277.108,A -85,B 0,C 180,E1 -4520.925,E2 -4520.925} C_VEL
LIN {X 0,Y 532.393,Z 264.591,A -85,B 0,C 180,E1 -4521.256,E2 -4521.256} C_VEL
LIN {X 0,Y 532.357,Z 264.168,A -85,B 0,C 180,E1 -4521.327,E2 -4521.327} C_VEL
LIN {X 0,Y 531.402,Z 262.246,A -85,B 0,C 180,E1 -4521.689,E2 -4521.689} C_VEL
LIN {X 0,Y 528.008,Z 259.724,A -85,B 0,C 180,E1 -4522.272,E2 -4522.272} C_VEL
LIN {X 0,Y 525.237,Z 258.397,A -85,B 0,C 180,E1 -4522.766,E2 -4522.766} C_VEL
LIN {X 0,Y 524.015,Z 257.89,A -85,B 0,C 180,E1 -4523.179,E2 -4523.179} C_VEL
LIN {X 0,Y 523.91,Z 257.851,A -85,B 0,C 180,E1 -4523.324,E2 -4523.324} C_VEL
LIN {X 0,Y 523.933,Z 257.847,A -85,B 0,C 180,E1 -4526.273,E2 -4526.273} C_VEL
LIN {X 0,Y 523.953,Z 257.842,A -85,B 0,C 180,E1 -4529.322,E2 -4529.322} C_VEL
LIN {X 0,Y 523.933,Z 257.843,A -85,B 0,C 180,E1 -4532.448,E2 -4532.448} C_VEL
LIN {X 0,Y 523.917,Z 257.844,A -85,B 0,C 180,E1 -4535.226,E2 -4535.226} C_VEL
LIN {X 0,Y 523.912,Z 257.849,A -85,B 0,C 180,E1 -4538.101,E2 -4538.101} C_VEL
LIN {X 0,Y 523.937,Z 257.841,A -85,B 0,C 180,E1 -4541.091,E2 -4541.091} C_VEL
LIN {X 0,Y 523.929,Z 257.845,A -85,B 0,C 180,E1 -4544.228,E2 -4544.228} C_VEL
LIN {X 0,Y 523.914,Z 257.844,A -85,B 0,C 180,E1 -4546.832,E2 -4546.832} C_VEL
LIN {X 0,Y 523.936,Z 257.841,A -85,B 0,C 180,E1 -4548.907,E2 -4548.907} C_VEL
LIN {X 0,Y 523.912,Z 257.851,A -85,B 0,C 180,E1 -4551.897,E2 -4551.897} C_VEL
LIN {X 0,Y 523.921,Z 257.843,A -85,B 0,C 180,E1 -4554.91,E2 -4554.91} C_VEL
LIN {X 0,Y 523.93,Z 257.85,A -85,B 0,C 180,E1 -4557.679,E2 -4557.679} C_VEL
LIN {X 0,Y 523.949,Z 257.839,A -85,B 0,C 180,E1 -4560.676,E2 -4560.676} C_VEL
LIN {X 0,Y 523.932,Z 257.851,A -85,B 0,C 180,E1 -4563.725,E2 -4563.725} C_VEL
LIN {X 0,Y 523.906,Z 257.846,A -85,B 0,C 180,E1 -4566.268,E2 -4566.268} C_VEL
LIN {X 0,Y 523.94,Z 257.84,A -85,B 0,C 180,E1 -4568.766,E2 -4568.766} C_VEL
LIN {X 0,Y 523.942,Z 257.843,A -85,B 0,C 180,E1 -4571.219,E2 -4571.219} C_VEL
LIN {X 0,Y 523.928,Z 257.851,A -85,B 0,C 180,E1 -4573.638,E2 -4573.638} C_VEL
LIN {X 0,Y 523.93,Z 257.845,A -85,B 0,C 180,E1 -4576.027,E2 -4576.027} C_VEL
LIN {X 0,Y 524.006,Z 257.833,A -85,B 0,C 180,E1 -4578.393,E2 -4578.393} C_VEL
LIN {X 0,Y 523.996,Z 257.841,A -85,B 0,C 180,E1 -4581.515,E2 -4581.515} C_VEL
LIN {X 0,Y 524.072,Z 257.824,A -85,B 0,C 180,E1 -4584.613,E2 -4584.613} C_VEL
LIN {X 0,Y 524.1,Z 257.828,A -85,B 0,C 180,E1 -4587.693,E2 -4587.693} C_VEL
LIN {X 0,Y 524.114,Z 257.819,A -85,B 0,C 180,E1 -4590.767,E2 -4590.767} C_VEL
LIN {X 0,Y 524.063,Z 257.828,A -85,B 0,C 180,E1 -4593.074,E2 -4593.074} C_VEL
LIN {X 0,Y 524.027,Z 257.831,A -85,B 0,C 180,E1 -4596.158,E2 -4596.158} C_VEL
LIN {X 0,Y 523.989,Z 257.834,A -85,B 0,C 180,E1 -4598.483,E2 -4598.483} C_VEL
LIN {X 0,Y 523.992,Z 257.839,A -85,B 0,C 180,E1 -4601.738,E2 -4601.738} C_VEL
LIN {X 0,Y 523.981,Z 257.838,A -85,B 0,C 180,E1 -4605.051,E2 -4605.051} C_VEL
LIN {X 0,Y 523.952,Z 257.841,A -85,B 0,C 180,E1 -4607.968,E2 -4607.968} C_VEL
LIN {X 0,Y 523.96,Z 257.838,A -85,B 0,C 180,E1 -4610.409,E2 -4610.409} C_VEL
LIN {X 0,Y 523.899,Z 257.848,A -85,B 0,C 180,E1 -4612.893,E2 -4612.893} C_VEL
LIN {X 0,Y 523.971,Z 257.838,A -85,B 0,C 180,E1 -4616.019,E2 -4616.019} C_VEL
LIN {X 0,Y 523.926,Z 257.844,A -85,B 0,C 180,E1 -4618.874,E2 -4618.874} C_VEL
LIN {X 0,Y 523.918,Z 257.85,A -85,B 0,C 180,E1 -4621.543,E2 -4621.543} C_VEL
LIN {X 0,Y 523.929,Z 257.842,A -85,B 0,C 180,E1 -4624.289,E2 -4624.289} C_VEL
LIN {X 0,Y 523.896,Z 257.852,A -85,B 0,C 180,E1 -4627.131,E2 -4627.131} C_VEL
LIN {X 0,Y 523.922,Z 257.843,A -85,B 0,C 180,E1 -4630.129,E2 -4630.129} C_VEL
LIN {X 0,Y 523.923,Z 257.843,A -85,B 0,C 180,E1 -4632.459,E2 -4632.459} C_VEL
LIN {X 0,Y 523.941,Z 257.849,A -85,B 0,C 180,E1 -4635.308,E2 -4635.308} C_VEL
LIN {X 0,Y 523.943,Z 257.842,A -85,B 0,C 180,E1 -4638.689,E2 -4638.689} C_VEL
LIN {X 0,Y 523.905,Z 257.851,A -85,B 0,C 180,E1 -4641.08,E2 -4641.08} C_VEL
LIN {X 0,Y 523.909,Z 257.846,A -85,B 0,C 180,E1 -4643.827,E2 -4643.827} C_VEL
LIN {X 0,Y 523.928,Z 257.844,A -85,B 0,C 180,E1 -4646.636,E2 -4646.636} C_VEL
LIN {X 0,Y 523.941,Z 257.847,A -85,B 0,C 180,E1 -4649.356,E2 -4649.356} C_VEL
LIN {X 0,Y 523.963,Z 257.837,A -85,B 0,C 180,E1 -4652.281,E2 -4652.281} C_VEL
LIN {X 0,Y 523.937,Z 257.842,A -85,B 0,C 180,E1 -4654.581,E2 -4654.581} C_VEL
LIN {X 0,Y 523.896,Z 257.855,A -85,B 0,C 180,E1 -4657.107,E2 -4657.107} C_VEL
LIN {X 0,Y 523.964,Z 257.838,A -85,B 0,C 180,E1 -4659.866,E2 -4659.866} C_VEL
LIN {X 0,Y 523.952,Z 257.844,A -85,B 0,C 180,E1 -4662.838,E2 -4662.838} C_VEL
LIN {X 0,Y 523.962,Z 257.845,A -85,B 0,C 180,E1 -4665.236,E2 -4665.236} C_VEL
LIN {X 0,Y 523.998,Z 257.834,A -85,B 0,C 180,E1 -4668.395,E2 -4668.395} C_VEL
LIN {X 0,Y 523.985,Z 257.838,A -85,B 0,C 180,E1 -4671.516,E2 -4671.516} C_VEL
LIN {X 0,Y 524.066,Z 257.828,A -85,B 0,C 180,E1 -4674.614,E2 -4674.614} C_VEL
LIN {X 0,Y 524.094,Z 257.822,A -85,B 0,C 180,E1 -4677.695,E2 -4677.695} C_VEL
LIN {X 0,Y 524.114,Z 257.824,A -85,B 0,C 180,E1 -4680.769,E2 -4680.769} C_VEL
LIN {X 0,Y 524.06,Z 257.834,A -85,B 0,C 180,E1 -4683.076,E2 -4683.076} C_VEL
LIN {X 0,Y 524.022,Z 257.83,A -85,B 0,C 180,E1 -4686.16,E2 -4686.16} C_VEL
LIN {X 0,Y 523.992,Z 257.836,A -85,B 0,C 180,E1 -4688.485,E2 -4688.485} C_VEL
LIN {X 0,Y 523.993,Z 257.834,A -85,B 0,C 180,E1 -4691.741,E2 -4691.741} C_VEL
LIN {X 0,Y 523.981,Z 257.843,A -85,B 0,C 180,E1 -4695.053,E2 -4695.053} C_VEL
LIN {X 0,Y 523.952,Z 257.839,A -85,B 0,C 180,E1 -4697.97,E2 -4697.97} C_VEL
LIN {X 0,Y 523.961,Z 257.84,A -85,B 0,C 180,E1 -4700.411,E2 -4700.411} C_VEL
LIN {X 0,Y 523.901,Z 257.855,A -85,B 0,C 180,E1 -4702.894,E2 -4702.894} C_VEL
LIN {X 0,Y 523.937,Z 257.843,A -85,B 0,C 180,E1 -4705.42,E2 -4705.42} C_VEL
LIN {X 0,Y 523.957,Z 257.838,A -85,B 0,C 180,E1 -4708,E2 -4708} C_VEL
LIN {X 0,Y 523.934,Z 257.85,A -85,B 0,C 180,E1 -4710.856,E2 -4710.856} C_VEL
LIN {X 0,Y 523.95,Z 257.839,A -85,B 0,C 180,E1 -4713.736,E2 -4713.736} C_VEL
LIN {X 0,Y 523.894,Z 257.85,A -85,B 0,C 180,E1 -4716.402,E2 -4716.402} C_VEL
LIN {X 0,Y 523.91,Z 257.849,A -85,B 0,C 180,E1 -4719.086,E2 -4719.086} C_VEL
LIN {X 0,Y 523.946,Z 257.841,A -85,B 0,C 180,E1 -4722.12,E2 -4722.12} C_VEL
LIN {X 0,Y 523.938,Z 257.842,A -85,B 0,C 180,E1 -4725.311,E2 -4725.311} C_VEL
LIN {X 0,Y 523.948,Z 257.848,A -85,B 0,C 180,E1 -4728.691,E2 -4728.691} C_VEL
LIN {X 0,Y 523.911,Z 257.849,A -85,B 0,C 180,E1 -4731.082,E2 -4731.082} C_VEL
LIN {X 0,Y 523.889,Z 257.847,A -85,B 0,C 180,E1 -4733.826,E2 -4733.826} C_VEL
LIN {X 0,Y 523.936,Z 257.848,A -85,B 0,C 180,E1 -4736.637,E2 -4736.637} C_VEL
LIN {X 0,Y 523.944,Z 257.845,A -85,B 0,C 180,E1 -4739.357,E2 -4739.357} C_VEL
LIN {X 0,Y 523.956,Z 257.891,A -85,B 0,C 180,E1 -4740.596,E2 -4740.596} C_VEL
LIN {X 0,Y 527.062,Z 270.516,A -85,B 0,C 180,E1 -4742.397,E2 -4742.397} C_VEL
LIN {X 0,Y 527.284,Z 273.9,A -85,B 0,C 180,E1 -4742.84,E2 -4742.84} C_VEL
LIN {X 0,Y 526.589,Z 295.944,A -85,B 0,C 180,E1 -4745.562,E2 -4745.562} C_VEL
LIN {X 0,Y 525.91,Z 320.119,A -85,B 0,C 180,E1 -4748.513,E2 -4748.513} C_VEL
LIN {X 0,Y 528.429,Z 335.232,A -85,B 0,C 180,E1 -4748.865,E2 -4748.865} C_VEL
LIN {X 0,Y 527.439,Z 470.91,A -85,B 0,C 180,E1 -4750.793,E2 -4750.793} C_VEL
LIN {X 0,Y 527.226,Z 491.014,A -85,B 0,C 180,E1 -4751.13,E2 -4751.13} C_VEL
LIN {X 0,Y 526.914,Z 506.862,A -85,B 0,C 180,E1 -4751.558,E2 -4751.558} C_VEL
LIN {X 0,Y 526.473,Z 521.746,A -85,B 0,C 180,E1 -4752.121,E2 -4752.121} C_VEL
LIN {X 0,Y 526.154,Z 535.759,A -85,B 0,C 180,E1 -4752.812,E2 -4752.812} C_VEL
LIN {X 0,Y 525.667,Z 548.673,A -85,B 0,C 180,E1 -4753.596,E2 -4753.596} C_VEL
LIN {X 0,Y 525.198,Z 562.026,A -85,B 0,C 180,E1 -4754.584,E2 -4754.584} C_VEL
LIN {X 0,Y 524.757,Z 574.071,A -85,B 0,C 180,E1 -4755.656,E2 -4755.656} C_VEL
LIN {X 0,Y 524.43,Z 585.162,A -85,B 0,C 180,E1 -4756.832,E2 -4756.832} C_VEL
LIN {X 0,Y 524.115,Z 594.555,A -85,B 0,C 180,E1 -4758.006,E2 -4758.006} C_VEL
LIN {X 0,Y 523.926,Z 603.745,A -85,B 0,C 180,E1 -4759.372,E2 -4759.372} C_VEL
LIN {X 0,Y 523.671,Z 611.348,A -85,B 0,C 180,E1 -4760.733,E2 -4760.733} C_VEL
LIN {X 0,Y 523.515,Z 618.445,A -85,B 0,C 180,E1 -4762.286,E2 -4762.286} C_VEL
LIN {X 0,Y 523.436,Z 624.017,A -85,B 0,C 180,E1 -4763.835,E2 -4763.835} C_VEL
LIN {X 0,Y 523.322,Z 628.221,A -85,B 0,C 180,E1 -4765.379,E2 -4765.379} C_VEL
LIN {X 0,Y 523.358,Z 631.166,A -85,B 0,C 180,E1 -4766.922,E2 -4766.922} C_VEL
LIN {X 0,Y 523.272,Z 632.905,A -85,B 0,C 180,E1 -4768.462,E2 -4768.462} C_VEL
LIN {X 0,Y 523.244,Z 633.498,A -85,B 0,C 180,E1 -4770.001,E2 -4770.001} C_VEL
LIN {X 0,Y 523.272,Z 632.901,A -85,B 0,C 180,E1 -4771.54,E2 -4771.54} C_VEL
LIN {X 0,Y 523.359,Z 631.158,A -85,B 0,C 180,E1 -4773.08,E2 -4773.08} C_VEL
LIN {X 0,Y 523.323,Z 628.211,A -85,B 0,C 180,E1 -4774.623,E2 -4774.623} C_VEL
LIN {X 0,Y 523.431,Z 624.002,A -85,B 0,C 180,E1 -4776.167,E2 -4776.167} C_VEL
LIN {X 0,Y 523.517,Z 618.405,A -85,B 0,C 180,E1 -4777.716,E2 -4777.716} C_VEL
LIN {X 0,Y 523.671,Z 611.264,A -85,B 0,C 180,E1 -4779.269,E2 -4779.269} C_VEL
LIN {X 0,Y 523.926,Z 603.612,A -85,B 0,C 180,E1 -4780.63,E2 -4780.63} C_VEL
LIN {X 0,Y 524.104,Z 594.324,A -85,B 0,C 180,E1 -4782.001,E2 -4782.001} C_VEL
LIN {X 0,Y 524.504,Z 583.171,A -85,B 0,C 180,E1 -4783.365,E2 -4783.365} C_VEL
LIN {X 0,Y 524.854,Z 571.634,A -85,B 0,C 180,E1 -4784.542,E2 -4784.542} C_VEL
LIN {X 0,Y 525.247,Z 559.819,A -85,B 0,C 180,E1 -4785.552,E2 -4785.552} C_VEL
LIN {X 0,Y 525.648,Z 546.409,A -85,B 0,C 180,E1 -4786.507,E2 -4786.507} C_VEL
LIN {X 0,Y 526.127,Z 532.883,A -85,B 0,C 180,E1 -4787.291,E2 -4787.291} C_VEL
LIN {X 0,Y 526.526,Z 519.197,A -85,B 0,C 180,E1 -4787.93,E2 -4787.93} C_VEL
LIN {X 0,Y 526.816,Z 504.146,A -85,B 0,C 180,E1 -4788.473,E2 -4788.473} C_VEL
LIN {X 0,Y 527.115,Z 488.577,A -85,B 0,C 180,E1 -4788.867,E2 -4788.867} C_VEL
LIN {X 0,Y 527.386,Z 458.819,A -85,B 0,C 180,E1 -4789.322,E2 -4789.322} C_VEL
LIN {X 0,Y 528.055,Z 374.597,A -85,B 0,C 180,E1 -4790.539,E2 -4790.539} C_VEL
LIN {X 0,Y 528.214,Z 333.554,A -85,B 0,C 180,E1 -4791.151,E2 -4791.151} C_VEL
LIN {X 0,Y 525.668,Z 318.694,A -85,B 0,C 180,E1 -4791.499,E2 -4791.499} C_VEL
LIN {X 0,Y 526.237,Z 295.789,A -85,B 0,C 180,E1 -4794.248,E2 -4794.248} C_VEL
LIN {X 0,Y 526.86,Z 273.642,A -85,B 0,C 180,E1 -4796.972,E2 -4796.972} C_VEL
LIN {X 0,Y 526.827,Z 270.248,A -85,B 0,C 180,E1 -4797.403,E2 -4797.403} C_VEL
LIN {X 0,Y 523.946,Z 257.849,A -85,B 0,C 180,E1 -4799.177,E2 -4799.177} C_VEL
LIN {X 0,Y 523.924,Z 257.851,A -85,B 0,C 180,E1 -4801.545,E2 -4801.545} C_VEL
LIN {X 0,Y 523.937,Z 257.846,A -85,B 0,C 180,E1 -4804.291,E2 -4804.291} C_VEL
LIN {X 0,Y 523.912,Z 257.853,A -85,B 0,C 180,E1 -4807.133,E2 -4807.133} C_VEL
LIN {X 0,Y 523.943,Z 257.843,A -85,B 0,C 180,E1 -4810.13,E2 -4810.13} C_VEL
LIN {X 0,Y 523.94,Z 257.846,A -85,B 0,C 180,E1 -4812.459,E2 -4812.459} C_VEL
LIN {X 0,Y 523.959,Z 257.843,A -85,B 0,C 180,E1 -4815.309,E2 -4815.309} C_VEL
LIN {X 0,Y 523.961,Z 257.846,A -85,B 0,C 180,E1 -4818.69,E2 -4818.69} C_VEL
